C03647=1132.728,344.800,-80.962,-177.361,10.889,149.504
C03648=1132.732,344.553,-80.928,-177.364,10.887,149.505
C03649=1132.736,344.305,-80.893,-177.367,10.884,149.505
C03650=1132.740,344.057,-80.858,-177.370,10.882,149.505
C03651=1132.744,343.810,-80.823,-177.374,10.879,149.505
C03652=1132.748,343.562,-80.789,-177.377,10.877,149.505
C03653=1132.752,343.315,-80.754,-177.380,10.874,149.506
C03654=1132.756,343.067,-80.719,-177.384,10.872,149.506
C03655=1132.760,342.820,-80.685,-177.387,10.869,149.506
C03656=1132.764,342.572,-80.650,-177.390,10.867,149.506
C03657=1132.768,342.325,-80.615,-177.393,10.864,149.506
C03658=1132.771,342.077,-80.581,-177.396,10.862,149.507
C03659=1132.776,341.830,-80.547,-177.400,10.859,149.507
C03660=1132.780,341.582,-80.512,-177.403,10.857,149.507
C03661=1132.784,341.334,-80.478,-177.406,10.854,149.507
C03662=1132.787,341.087,-80.443,-177.409,10.851,149.507
C03663=1132.791,340.840,-80.409,-177.413,10.849,149.508
C03664=1132.795,340.592,-80.374,-177.416,10.847,149.508
C03665=1132.800,340.344,-80.339,-177.419,10.844,149.508
C03666=1132.803,340.097,-80.305,-177.422,10.841,149.508
C03667=1132.808,339.849,-80.271,-177.426,10.839,149.508
C03668=1132.811,339.602,-80.237,-177.429,10.836,149.509
C03669=1132.815,339.354,-80.202,-177.432,10.834,149.509
C03670=1132.819,339.107,-80.168,-177.435,10.832,149.509
C03671=1132.823,338.859,-80.133,-177.438,10.829,149.509
C03672=1132.827,338.612,-80.099,-177.442,10.826,149.509
C03673=1132.831,338.363,-80.065,-177.445,10.824,149.510
C03674=1132.835,338.116,-80.031,-177.448,10.821,149.510
C03675=1132.840,337.868,-79.997,-177.452,10.819,149.510
C03676=1132.843,337.620,-79.963,-177.455,10.816,149.510
C03677=1132.848,337.373,-79.928,-177.458,10.814,149.510
C03678=1132.851,337.125,-79.894,-177.461,10.811,149.511
C03679=1132.855,336.878,-79.860,-177.465,10.809,149.511
C03680=1132.859,336.630,-79.825,-177.468,10.806,149.511
C03681=1132.863,336.383,-79.791,-177.471,10.804,149.511
C03682=1132.867,336.135,-79.758,-177.473,10.802,149.511
C03683=1132.870,335.887,-79.723,-177.477,10.799,149.512
C03684=1132.875,335.674,-79.694,-177.480,10.797,149.512
C03685=1132.877,335.461,-79.664,-177.482,10.795,149.512
C03686=1132.881,335.248,-79.635,-177.486,10.793,149.512
C03687=1132.885,335.034,-79.605,-177.488,10.791,149.512
C03688=1132.888,334.821,-79.576,-177.491,10.788,149.513
C03689=1132.892,334.608,-79.547,-177.494,10.786,149.513
C03690=1132.895,334.395,-79.518,-177.496,10.784,149.513
C03691=1132.899,334.182,-79.489,-177.499,10.782,149.513
C03692=1132.902,333.934,-79.454,-177.503,10.779,149.513
C03693=1132.906,333.687,-79.421,-177.506,10.777,149.513
C03694=1132.911,333.439,-79.387,-177.509,10.774,149.514
C03695=1132.914,333.191,-79.353,-177.512,10.772,149.514
C03696=1132.918,332.943,-79.319,-177.515,10.769,149.514
C03697=1132.923,332.696,-79.285,-177.519,10.767,149.514
C03698=1132.926,332.448,-79.251,-177.522,10.764,149.514
C03699=1132.930,332.200,-79.218,-177.525,10.761,149.515
C03700=1132.934,331.953,-79.184,-177.528,10.759,149.515
C03701=1132.938,331.704,-79.150,-177.531,10.757,149.515
C03702=1132.942,331.457,-79.116,-177.534,10.754,149.515
C03703=1132.946,331.209,-79.083,-177.537,10.752,149.515
C03704=1132.950,330.962,-79.049,-177.541,10.750,149.516
C03705=1132.954,330.714,-79.015,-177.544,10.747,149.516
C03706=1132.958,330.466,-78.981,-177.547,10.744,149.516
C03707=1132.962,330.219,-78.948,-177.550,10.742,149.516
C03708=1132.966,329.972,-78.914,-177.553,10.739,149.516
C03709=1132.970,329.723,-78.880,-177.557,10.737,149.517
C03710=1132.974,329.476,-78.846,-177.560,10.734,149.517
C03711=1132.978,329.228,-78.813,-177.563,10.732,149.517
C03712=1132.982,328.980,-78.779,-177.566,10.729,149.517
C03713=1132.986,328.732,-78.745,-177.569,10.727,149.517
C03714=1132.990,328.485,-78.712,-177.573,10.724,149.517
C03715=1132.994,328.238,-78.678,-177.576,10.722,149.518
C03716=1132.998,327.990,-78.644,-177.579,10.719,149.518
C03717=1133.003,327.742,-78.611,-177.582,10.716,149.518
C03718=1133.006,327.494,-78.577,-177.585,10.714,149.518
C03719=1133.010,327.246,-78.544,-177.589,10.712,149.519
C03720=1133.014,326.999,-78.511,-177.592,10.709,149.519
C03721=1133.018,326.751,-78.478,-177.595,10.706,149.519
C03722=1133.022,326.504,-78.444,-177.598,10.704,149.519
C03723=1133.026,326.256,-78.411,-177.602,10.701,149.519
C03724=1133.030,326.008,-78.377,-177.605,10.699,149.519
C03725=1133.034,325.760,-78.344,-177.608,10.696,149.520
C03726=1133.038,325.512,-78.311,-177.611,10.694,149.520
C03727=1133.042,325.265,-78.277,-177.614,10.691,149.520
C03728=1133.046,325.017,-78.244,-177.617,10.689,149.520
C03729=1133.050,324.770,-78.211,-177.620,10.687,149.521
C03730=1133.054,324.521,-78.177,-177.623,10.684,149.521
C03731=1133.058,324.273,-78.144,-177.626,10.682,149.521
C03732=1133.062,324.026,-78.111,-177.630,10.679,149.521
C03733=1133.066,323.778,-78.078,-177.633,10.676,149.521
C03734=1133.070,323.530,-78.044,-177.636,10.674,149.521
C03735=1133.074,323.283,-78.010,-177.639,10.672,149.522
C03736=1133.078,323.035,-77.977,-177.643,10.669,149.522
C03737=1133.082,322.788,-77.944,-177.646,10.666,149.522
C03738=1133.086,322.540,-77.911,-177.649,10.664,149.522
C03739=1133.090,322.291,-77.877,-177.652,10.661,149.522
C03740=1133.094,322.078,-77.849,-177.655,10.659,149.523
C03741=1133.097,321.865,-77.820,-177.657,10.657,149.523
C03742=1133.100,321.652,-77.793,-177.660,10.655,149.523
C03743=1133.104,321.438,-77.764,-177.663,10.652,149.523
C03744=1133.107,321.225,-77.735,-177.666,10.651,149.523
C03745=1133.111,321.011,-77.707,-177.669,10.648,149.523
C03746=1133.115,320.798,-77.678,-177.671,10.646,149.524
C03747=1133.118,320.585,-77.650,-177.674,10.644,149.524
C03748=1133.123,320.337,-77.617,-177.677,10.642,149.524
C03749=1133.125,320.089,-77.584,-177.680,10.639,149.524
C03750=1133.129,319.841,-77.551,-177.683,10.637,149.524
C03751=1133.134,319.594,-77.518,-177.687,10.634,149.525
C03752=1133.138,319.345,-77.485,-177.690,10.631,149.525
C03753=1133.142,319.098,-77.452,-177.693,10.629,149.525
C03754=1133.146,318.850,-77.420,-177.696,10.626,149.525
C03755=1133.150,318.602,-77.387,-177.699,10.624,149.525
C03756=1133.154,318.355,-77.353,-177.702,10.621,149.525
C03757=1133.158,318.106,-77.321,-177.705,10.618,149.525
C03758=1133.162,317.859,-77.288,-177.709,10.616,149.526
C03759=1133.166,317.611,-77.255,-177.712,10.614,149.526
C03760=1133.170,317.363,-77.222,-177.715,10.611,149.526
C03761=1133.174,317.115,-77.190,-177.718,10.608,149.526
C03762=1133.178,316.868,-77.157,-177.722,10.606,149.527
C03763=1133.182,316.620,-77.124,-177.725,10.603,149.527
C03764=1133.186,316.372,-77.091,-177.728,10.601,149.527
C03765=1133.191,316.125,-77.059,-177.731,10.598,149.527
C03766=1133.195,315.877,-77.026,-177.733,10.596,149.527
C03767=1133.199,315.629,-76.994,-177.737,10.594,149.527
C03768=1133.203,315.381,-76.961,-177.740,10.591,149.528
C03769=1133.207,315.133,-76.929,-177.743,10.589,149.528
C03770=1133.211,314.885,-76.896,-177.746,10.586,149.528
C03771=1133.215,314.638,-76.862,-177.749,10.583,149.528
C03772=1133.219,314.389,-76.831,-177.753,10.581,149.528
C03773=1133.223,314.142,-76.797,-177.756,10.578,149.528
C03774=1133.227,313.894,-76.766,-177.759,10.576,149.529
C03775=1133.231,313.646,-76.732,-177.762,10.573,149.529
C03776=1133.235,313.398,-76.700,-177.765,10.571,149.529
C03777=1133.239,313.151,-76.668,-177.768,10.568,149.529
C03778=1133.244,312.903,-76.635,-177.771,10.565,149.529
C03779=1133.247,312.655,-76.603,-177.775,10.563,149.530
C03780=1133.252,312.407,-76.570,-177.778,10.560,149.530
C03781=1133.256,312.158,-76.538,-177.781,10.558,149.530
C03782=1133.259,311.911,-76.505,-177.784,10.555,149.530
C03783=1133.264,311.663,-76.473,-177.787,10.552,149.530
C03784=1133.268,311.416,-76.441,-177.791,10.550,149.531
C03785=1133.272,311.168,-76.408,-177.794,10.548,149.531
C03786=1133.276,310.920,-76.376,-177.796,10.546,149.531
C03787=1133.280,310.672,-76.343,-177.800,10.543,149.531
C03788=1133.284,310.424,-76.311,-177.802,10.540,149.531
C03789=1133.288,310.175,-76.279,-177.806,10.538,149.532
C03790=1133.292,309.929,-76.247,-177.809,10.536,149.532
C03791=1133.297,309.680,-76.214,-177.812,10.533,149.532
C03792=1133.300,309.432,-76.182,-177.815,10.530,149.532
C03793=1133.305,309.184,-76.150,-177.818,10.528,149.532
C03794=1133.308,308.937,-76.117,-177.822,10.525,149.532
C03795=1133.313,308.689,-76.086,-177.825,10.522,149.533
C03796=1133.316,308.476,-76.058,-177.827,10.521,149.533
C03797=1133.320,308.262,-76.031,-177.830,10.518,149.533
C03798=1133.324,308.048,-76.003,-177.833,10.516,149.533
C03799=1133.327,307.835,-75.975,-177.836,10.514,149.533
C03800=1133.331,307.621,-75.948,-177.838,10.512,149.533
C03801=1133.334,307.408,-75.920,-177.841,10.510,149.534
C03802=1133.338,307.194,-75.892,-177.844,10.507,149.534
C03803=1133.341,306.981,-75.864,-177.846,10.505,149.534
C03804=1133.345,306.733,-75.832,-177.849,10.503,149.534
C03805=1133.349,306.485,-75.800,-177.852,10.500,149.534
C03806=1133.353,306.237,-75.768,-177.856,10.497,149.534
C03807=1133.358,305.989,-75.736,-177.859,10.495,149.535
C03808=1133.361,305.741,-75.704,-177.862,10.492,149.535
C03809=1133.365,305.493,-75.673,-177.865,10.490,149.535
C03810=1133.370,305.245,-75.640,-177.868,10.487,149.535
C03811=1133.374,304.997,-75.609,-177.872,10.485,149.535
C03812=1133.378,304.749,-75.577,-177.874,10.482,149.535
C03813=1133.382,304.501,-75.544,-177.878,10.479,149.536
C03814=1133.386,304.254,-75.513,-177.880,10.477,149.536
C03815=1133.390,304.006,-75.481,-177.883,10.475,149.536
C03816=1133.395,303.757,-75.449,-177.886,10.472,149.536
C03817=1133.399,303.510,-75.417,-177.890,10.470,149.536
C03818=1133.403,303.262,-75.385,-177.893,10.467,149.537
C03819=1133.406,303.014,-75.353,-177.896,10.465,149.537
C03820=1133.412,302.766,-75.322,-177.899,10.462,149.537
C03821=1133.415,302.518,-75.290,-177.902,10.459,149.537
C03822=1133.420,302.270,-75.259,-177.906,10.457,149.537
C03823=1133.423,302.022,-75.227,-177.909,10.454,149.538
C03824=1133.427,301.774,-75.195,-177.912,10.452,149.538
C03825=1133.432,301.526,-75.163,-177.915,10.449,149.538
C03826=1133.436,301.278,-75.132,-177.918,10.447,149.538
C03827=1133.440,301.030,-75.100,-177.921,10.444,149.538
C03828=1133.444,300.782,-75.068,-177.924,10.441,149.538
C03829=1133.448,300.534,-75.037,-177.927,10.439,149.539
C03830=1133.452,300.286,-75.006,-177.930,10.437,149.539
C03831=1133.457,300.038,-74.973,-177.933,10.434,149.539
C03832=1133.461,299.790,-74.942,-177.936,10.432,149.539
C03833=1133.465,299.543,-74.910,-177.939,10.429,149.539
C03834=1133.469,299.294,-74.879,-177.943,10.427,149.540
C03835=1133.473,299.047,-74.847,-177.945,10.424,149.540
C03836=1133.477,298.799,-74.816,-177.949,10.421,149.540
C03837=1133.482,298.551,-74.785,-177.952,10.419,149.540
C03838=1133.485,298.303,-74.753,-177.955,10.416,149.540
C03839=1133.490,298.055,-74.722,-177.958,10.414,149.541
C03840=1133.494,297.807,-74.690,-177.961,10.411,149.541
C03841=1133.497,297.559,-74.659,-177.965,10.409,149.541
C03842=1133.502,297.311,-74.628,-177.968,10.406,149.541
C03843=1133.506,297.063,-74.596,-177.971,10.403,149.541
C03844=1133.510,296.815,-74.565,-177.973,10.401,149.541
C03845=1133.514,296.567,-74.533,-177.977,10.399,149.542
C03846=1133.518,296.319,-74.503,-177.980,10.396,149.542
C03847=1133.522,296.071,-74.471,-177.983,10.394,149.542
C03848=1133.527,295.823,-74.440,-177.986,10.391,149.542
C03849=1133.531,295.575,-74.408,-177.989,10.389,149.542
C03850=1133.535,295.327,-74.377,-177.992,10.386,149.542
C03851=1133.539,295.079,-74.346,-177.995,10.383,149.543
C03852=1133.542,294.865,-74.319,-177.998,10.381,149.543
C03853=1133.546,294.652,-74.292,-178.001,10.379,149.543
C03854=1133.550,294.438,-74.265,-178.003,10.377,149.543
C03855=1133.553,294.224,-74.238,-178.006,10.375,149.543
C03856=1133.557,294.010,-74.211,-178.009,10.372,149.543
C03857=1133.561,293.797,-74.185,-178.011,10.370,149.544
C03858=1133.565,293.583,-74.158,-178.014,10.368,149.544
C03859=1133.568,293.369,-74.131,-178.017,10.366,149.544
C03860=1133.573,293.121,-74.100,-178.019,10.363,149.544
C03861=1133.576,292.874,-74.069,-178.023,10.361,149.544
C03862=1133.580,292.626,-74.038,-178.026,10.358,149.544
C03863=1133.584,292.377,-74.007,-178.029,10.356,149.545
C03864=1133.588,292.130,-73.975,-178.032,10.353,149.545
C03865=1133.592,291.881,-73.944,-178.035,10.350,149.545
C03866=1133.597,291.633,-73.914,-178.038,10.348,149.545
C03867=1133.600,291.385,-73.883,-178.041,10.346,149.545
C03868=1133.605,291.137,-73.852,-178.044,10.343,149.545
C03869=1133.609,290.889,-73.821,-178.047,10.341,149.546
C03870=1133.613,290.641,-73.790,-178.050,10.338,149.546
C03871=1133.618,290.393,-73.759,-178.053,10.335,149.546
C03872=1133.622,290.145,-73.729,-178.056,10.333,149.546
C03873=1133.625,289.897,-73.697,-178.059,10.330,149.546
C03874=1133.630,289.649,-73.666,-178.063,10.328,149.547
C03875=1133.634,289.400,-73.635,-178.066,10.325,149.547
C03876=1133.638,289.153,-73.605,-178.069,10.322,149.547
C03877=1133.643,288.905,-73.574,-178.072,10.320,149.547
C03878=1133.647,288.656,-73.543,-178.075,10.318,149.547
C03879=1133.650,288.408,-73.513,-178.078,10.315,149.547
C03880=1133.655,288.161,-73.482,-178.081,10.313,149.548
C03881=1133.659,287.912,-73.451,-178.084,10.310,149.548
C03882=1133.664,287.664,-73.420,-178.087,10.307,149.548
C03883=1133.668,287.416,-73.390,-178.090,10.305,149.548
C03884=1133.672,287.168,-73.359,-178.093,10.302,149.548
C03885=1133.676,286.920,-73.328,-178.096,10.300,149.549
C03886=1133.680,286.672,-73.298,-178.099,10.297,149.549
C03887=1133.684,286.423,-73.267,-178.103,10.295,149.549
C03888=1133.688,286.176,-73.237,-178.106,10.292,149.549
C03889=1133.693,285.928,-73.206,-178.109,10.289,149.549
C03890=1133.697,285.680,-73.175,-178.111,10.287,149.549
C03891=1133.700,285.431,-73.144,-178.114,10.285,149.550
C03892=1133.705,285.183,-73.114,-178.118,10.282,149.550
C03893=1133.709,284.936,-73.084,-178.121,10.279,149.550
C03894=1133.714,284.688,-73.053,-178.124,10.277,149.550
C03895=1133.718,284.439,-73.022,-178.127,10.274,149.550
C03896=1133.722,284.191,-72.992,-178.130,10.272,149.551
C03897=1133.726,283.943,-72.961,-178.133,10.269,149.551
C03898=1133.730,283.695,-72.931,-178.136,10.267,149.551
C03899=1133.734,283.447,-72.900,-178.139,10.264,149.551
C03900=1133.738,283.198,-72.871,-178.142,10.261,149.551
C03901=1133.743,282.950,-72.840,-178.145,10.259,149.551
C03902=1133.747,282.703,-72.810,-178.148,10.257,149.552
C03903=1133.751,282.454,-72.779,-178.151,10.254,149.552
C03904=1133.755,282.206,-72.749,-178.154,10.252,149.552
C03905=1133.760,281.958,-72.718,-178.158,10.249,149.552
C03906=1133.764,281.710,-72.688,-178.161,10.246,149.552
C03907=1133.768,281.462,-72.657,-178.163,10.244,149.552
C03908=1133.772,281.248,-72.631,-178.167,10.241,149.553
C03909=1133.776,281.034,-72.606,-178.170,10.239,149.553
C03910=1133.779,280.821,-72.579,-178.173,10.236,149.553
C03911=1133.783,280.606,-72.553,-178.176,10.234,149.553
C03912=1133.786,280.393,-72.528,-178.179,10.231,149.553
C03913=1133.790,280.179,-72.501,-178.183,10.228,149.554
C03914=1133.794,279.965,-72.475,-178.185,10.226,149.554
C03915=1133.797,279.751,-72.450,-178.188,10.224,149.554
C03916=1133.801,279.503,-72.419,-178.192,10.221,149.554
C03917=1133.806,279.255,-72.390,-178.195,10.218,149.554
C03918=1133.810,279.007,-72.359,-178.199,10.215,149.555
C03919=1133.814,278.759,-72.329,-178.203,10.213,149.555
C03920=1133.818,278.511,-72.299,-178.206,10.209,149.555
C03921=1133.822,278.262,-72.269,-178.210,10.207,149.555
C03922=1133.827,278.014,-72.239,-178.212,10.204,149.555
C03923=1133.831,277.766,-72.209,-178.216,10.201,149.556
C03924=1133.835,277.518,-72.179,-178.220,10.198,149.556
C03925=1133.839,277.270,-72.149,-178.223,10.195,149.556
C03926=1133.844,277.021,-72.119,-178.227,10.192,149.556
C03927=1133.848,276.774,-72.089,-178.230,10.189,149.557
C03928=1133.852,276.525,-72.060,-178.233,10.187,149.557
C03929=1133.856,276.277,-72.029,-178.237,10.184,149.557
C03930=1133.861,276.029,-72.000,-178.240,10.181,149.557
C03931=1133.865,275.781,-71.970,-178.243,10.178,149.557
C03932=1133.869,275.533,-71.940,-178.246,10.176,149.557
C03933=1133.873,275.284,-71.910,-178.249,10.173,149.557
C03934=1133.877,275.036,-71.880,-178.253,10.170,149.558
C03935=1133.881,274.787,-71.851,-178.256,10.167,149.558
C03936=1133.885,274.540,-71.820,-178.259,10.164,149.558
C03937=1133.889,274.291,-71.791,-178.262,10.161,149.558
C03938=1133.894,274.043,-71.762,-178.265,10.159,149.558
C03939=1133.898,273.795,-71.732,-178.268,10.156,149.558
C03940=1133.903,273.546,-71.702,-178.271,10.153,149.559
C03941=1133.906,273.299,-71.672,-178.274,10.151,149.559
C03942=1133.911,273.050,-71.642,-178.277,10.148,149.559
C03943=1133.915,272.802,-71.613,-178.280,10.146,149.559
C03944=1133.919,272.554,-71.584,-178.283,10.143,149.559
C03945=1133.923,272.306,-71.554,-178.286,10.140,149.559
C03946=1133.927,272.057,-71.525,-178.289,10.137,149.559
C03947=1133.932,271.809,-71.495,-178.292,10.135,149.559
C03948=1133.937,271.561,-71.466,-178.295,10.132,149.560
C03949=1133.941,271.314,-71.435,-178.297,10.130,149.560
C03950=1133.945,271.065,-71.406,-178.300,10.127,149.560
C03951=1133.949,270.817,-71.376,-178.303,10.124,149.560
C03952=1133.954,270.569,-71.347,-178.306,10.121,149.560
C03953=1133.958,270.321,-71.318,-178.309,10.119,149.560
C03954=1133.962,270.072,-71.288,-178.311,10.117,149.560
C03955=1133.966,269.824,-71.259,-178.314,10.114,149.560
C03956=1133.970,269.576,-71.229,-178.317,10.111,149.560
C03957=1133.974,269.327,-71.200,-178.319,10.109,149.561
C03958=1133.979,269.079,-71.170,-178.322,10.107,149.561
C03959=1133.983,268.830,-71.142,-178.325,10.104,149.561
C03960=1133.987,268.582,-71.112,-178.327,10.102,149.561
C03961=1133.992,268.334,-71.083,-178.330,10.099,149.561
C03962=1133.996,268.086,-71.054,-178.333,10.097,149.561
C03963=1134.000,267.838,-71.024,-178.335,10.094,149.561
C03964=1134.003,267.624,-70.999,-178.338,10.092,149.561
C03965=1134.007,267.410,-70.974,-178.340,10.090,149.561
C03966=1134.012,267.196,-70.948,-178.342,10.088,149.561
C03967=1134.015,266.982,-70.923,-178.344,10.086,149.561
C03968=1134.018,266.768,-70.898,-178.346,10.084,149.561
C03969=1134.023,266.554,-70.873,-178.349,10.082,149.562
C03970=1134.026,266.341,-70.847,-178.351,10.080,149.562
C03971=1134.030,266.126,-70.822,-178.353,10.077,149.562
C03972=1134.034,265.878,-70.793,-178.355,10.075,149.562
C03973=1134.039,265.630,-70.764,-178.357,10.073,149.562
C03974=1134.043,265.382,-70.734,-178.360,10.071,149.562
C03975=1134.047,265.133,-70.706,-178.362,10.068,149.562
C03976=1134.051,264.885,-70.677,-178.365,10.066,149.562
C03977=1134.055,264.637,-70.647,-178.367,10.064,149.562
C03978=1134.059,264.388,-70.618,-178.370,10.062,149.562
C03979=1134.064,264.140,-70.590,-178.374,10.058,149.563
C03980=1134.068,263.892,-70.560,-178.378,10.055,149.563
C03981=1134.072,263.644,-70.531,-178.382,10.052,149.563
C03982=1134.077,263.395,-70.502,-178.386,10.049,149.563
C03983=1134.080,263.147,-70.473,-178.390,10.046,149.564
C03984=1134.085,262.899,-70.444,-178.394,10.043,149.564
C03985=1134.090,262.650,-70.415,-178.397,10.039,149.564
C03986=1134.094,262.402,-70.386,-178.401,10.036,149.564
C03987=1134.098,262.154,-70.358,-178.405,10.033,149.565
C03988=1134.102,261.906,-70.329,-178.409,10.029,149.565
C03989=1134.107,261.657,-70.300,-178.413,10.026,149.565
C03990=1134.111,261.409,-70.270,-178.417,10.023,149.565
C03991=1134.115,261.161,-70.243,-178.420,10.019,149.565
C03992=1134.120,260.913,-70.213,-178.424,10.017,149.566
C03993=1134.124,260.664,-70.184,-178.427,10.013,149.566
C03994=1134.127,260.416,-70.156,-178.431,10.010,149.566
C03995=1134.133,260.168,-70.127,-178.434,10.007,149.566
C03996=1134.137,259.919,-70.098,-178.438,10.004,149.566
C03997=1134.140,259.671,-70.070,-178.442,10.001,149.567
C03998=1134.146,259.423,-70.041,-178.445,9.998,149.567
C03999=1134.150,259.174,-70.012,-178.448,9.994,149.567
C04000=1134.154,258.926,-69.984,-178.452,9.992,149.567
C04001=1134.159,258.678,-69.955,-178.455,9.988,149.567
C04002=1134.162,258.430,-69.926,-178.458,9.986,149.567
C04003=1134.167,258.181,-69.898,-178.461,9.983,149.567
C04004=1134.172,257.933,-69.869,-178.465,9.979,149.567
C04005=1134.175,257.685,-69.840,-178.468,9.977,149.568
C04006=1134.180,257.436,-69.812,-178.471,9.974,149.568
C04007=1134.184,257.188,-69.784,-178.474,9.971,149.568
C04008=1134.188,256.939,-69.755,-178.477,9.968,149.568
C04009=1134.192,256.691,-69.726,-178.480,9.965,149.568
C04010=1134.197,256.443,-69.698,-178.483,9.962,149.568
C04011=1134.201,256.194,-69.670,-178.486,9.959,149.568
C04012=1134.206,255.946,-69.641,-178.489,9.956,149.568
C04013=1134.210,255.698,-69.613,-178.488,9.956,149.568
C04014=1134.214,255.450,-69.584,-178.486,9.956,149.567
C04015=1134.218,255.201,-69.556,-178.485,9.955,149.567
C04016=1134.223,254.952,-69.527,-178.484,9.955,149.567
C04017=1134.227,254.705,-69.500,-178.484,9.954,149.566
C04018=1134.231,254.456,-69.471,-178.484,9.953,149.566
C04019=1134.236,254.208,-69.443,-178.484,9.952,149.566
C04020=1134.239,253.993,-69.418,-178.484,9.951,149.566
C04021=1134.243,253.780,-69.393,-178.485,9.950,149.566
C04022=1134.246,253.566,-69.369,-178.486,9.949,149.566
C04023=1134.250,253.352,-69.344,-178.487,9.947,149.566
C04024=1134.254,253.138,-69.320,-178.489,9.946,149.566
C04025=1134.258,252.923,-69.295,-178.490,9.944,149.566
C04026=1134.262,252.709,-69.271,-178.492,9.943,149.566
C04027=1134.266,252.495,-69.246,-178.494,9.941,149.566
C04028=1134.270,252.247,-69.218,-178.496,9.939,149.566
C04029=1134.273,251.998,-69.190,-178.499,9.936,149.566
C04030=1134.278,251.750,-69.162,-178.503,9.934,149.566
C04031=1134.282,251.501,-69.133,-178.506,9.930,149.567
C04032=1134.287,251.253,-69.105,-178.509,9.928,149.567
C04033=1134.291,251.005,-69.077,-178.514,9.924,149.567
C04034=1134.296,250.757,-69.049,-178.518,9.921,149.568
C04035=1134.300,250.508,-69.020,-178.523,9.917,149.568
C04036=1134.304,250.260,-68.993,-178.528,9.914,149.568
C04037=1134.309,250.011,-68.964,-178.533,9.910,149.569
C04038=1134.313,249.763,-68.936,-178.539,9.906,149.569
C04039=1134.317,249.515,-68.908,-178.545,9.901,149.570
C04040=1134.322,249.267,-68.880,-178.551,9.897,149.570
C04041=1134.326,249.018,-68.851,-178.558,9.891,149.571
C04042=1134.330,248.770,-68.824,-178.564,9.887,149.571
C04043=1134.334,248.521,-68.796,-178.572,9.881,149.572
C04044=1134.339,248.273,-68.768,-178.579,9.876,149.573
C04045=1134.343,248.024,-68.740,-178.586,9.870,149.573
C04046=1134.347,247.776,-68.712,-178.595,9.864,149.574
C04047=1134.352,247.528,-68.685,-178.603,9.858,149.575
C04048=1134.356,247.279,-68.657,-178.607,9.854,149.575
C04049=1134.361,247.031,-68.628,-178.608,9.852,149.575
C04050=1134.365,246.782,-68.601,-178.609,9.850,149.574
C04051=1134.369,246.534,-68.573,-178.610,9.848,149.574
C04052=1134.374,246.285,-68.546,-178.611,9.846,149.574
C04053=1134.377,246.037,-68.518,-178.613,9.844,149.574
C04054=1134.382,245.789,-68.490,-178.614,9.842,149.574
C04055=1134.386,245.540,-68.463,-178.614,9.840,149.573
C04056=1134.391,245.292,-68.434,-178.616,9.838,149.573
C04057=1134.396,245.043,-68.407,-178.617,9.836,149.573
C04058=1134.400,244.795,-68.380,-178.618,9.834,149.573
C04059=1134.404,244.546,-68.352,-178.619,9.832,149.573
C04060=1134.408,244.298,-68.324,-178.621,9.830,149.573
C04061=1134.412,244.049,-68.297,-178.622,9.828,149.573
C04062=1134.417,243.801,-68.269,-178.624,9.826,149.573
C04063=1134.421,243.553,-68.241,-178.625,9.824,149.573
C04064=1134.425,243.304,-68.214,-178.627,9.822,149.572
C04065=1134.430,243.056,-68.186,-178.629,9.819,149.572
C04066=1134.434,242.808,-68.159,-178.630,9.818,149.572
C04067=1134.438,242.559,-68.131,-178.632,9.816,149.572
C04068=1134.443,242.311,-68.104,-178.634,9.813,149.572
C04069=1134.447,242.062,-68.077,-178.636,9.811,149.572
C04070=1134.452,241.814,-68.048,-178.638,9.809,149.572
C04071=1134.456,241.565,-68.021,-178.640,9.806,149.572
C04072=1134.461,241.317,-67.993,-178.642,9.804,149.572
C04073=1134.465,241.068,-67.966,-178.644,9.802,149.572
C04074=1134.469,240.820,-67.938,-178.646,9.800,149.572
C04075=1134.474,240.571,-67.911,-178.648,9.797,149.572
C04076=1134.478,240.291,-67.880,-178.650,9.795,149.572
C04077=1134.484,240.010,-67.849,-178.653,9.792,149.572
C04078=1134.488,239.730,-67.819,-178.655,9.789,149.572
C04079=1134.493,239.450,-67.787,-178.657,9.787,149.572
C04080=1134.498,239.201,-67.760,-178.660,9.784,149.572
C04081=1134.502,238.952,-67.733,-178.662,9.782,149.572
C04082=1134.506,238.704,-67.705,-178.665,9.780,149.572
C04083=1134.511,238.456,-67.678,-178.667,9.777,149.573
C04084=1134.516,238.207,-67.651,-178.670,9.774,149.572
C04085=1134.520,237.958,-67.623,-178.672,9.772,149.573
C04086=1134.524,237.710,-67.596,-178.675,9.769,149.573
C04087=1134.529,237.462,-67.569,-178.677,9.767,149.573
C04088=1134.533,237.213,-67.541,-178.680,9.764,149.573
C04089=1134.536,236.965,-67.514,-178.683,9.762,149.573
C04090=1134.541,236.716,-67.487,-178.686,9.759,149.573
C04091=1134.546,236.468,-67.460,-178.689,9.756,149.573
C04092=1134.550,236.219,-67.433,-178.692,9.753,149.573
C04093=1134.554,235.970,-67.405,-178.695,9.751,149.573
C04094=1134.559,235.722,-67.378,-178.698,9.748,149.574
C04095=1134.563,235.474,-67.350,-178.701,9.745,149.574
C04096=1134.567,235.226,-67.324,-178.704,9.742,149.574
C04097=1134.572,234.977,-67.297,-178.707,9.740,149.574
C04098=1134.577,234.729,-67.270,-178.710,9.737,149.574
C04099=1134.581,234.480,-67.242,-178.713,9.734,149.574
C04100=1134.585,234.231,-67.215,-178.716,9.731,149.574
C04101=1134.589,233.983,-67.189,-178.719,9.728,149.574
C04102=1134.594,233.734,-67.162,-178.723,9.725,149.575
C04103=1134.598,233.486,-67.135,-178.726,9.722,149.575
C04104=1134.603,233.237,-67.108,-178.730,9.718,149.575
C04105=1134.606,232.988,-67.081,-178.733,9.716,149.575
C04106=1134.611,232.740,-67.054,-178.737,9.713,149.575
C04107=1134.616,232.491,-67.027,-178.740,9.709,149.576
C04108=1134.635,231.404,-66.912,-177.831,7.908,148.890
C04109=1134.639,231.186,-66.889,-177.834,7.905,148.890
C04110=1134.643,230.967,-66.866,-177.836,7.903,148.890
C04111=1134.647,230.748,-66.843,-177.839,7.900,148.890
C04112=1134.651,230.500,-66.817,-177.842,7.897,148.890
C04113=1134.656,230.251,-66.790,-177.845,7.894,148.890
C04114=1134.660,230.003,-66.764,-177.847,7.891,148.890
C04115=1134.664,229.754,-66.738,-177.850,7.888,148.890
C04116=1134.669,229.506,-66.711,-177.853,7.885,148.891
C04117=1134.673,229.257,-66.685,-177.856,7.882,148.891
C04118=1134.678,229.008,-66.658,-177.858,7.880,148.891
C04119=1134.682,228.760,-66.632,-177.861,7.877,148.891
C04120=1134.687,228.512,-66.606,-177.864,7.874,148.891
C04121=1134.692,228.263,-66.580,-177.866,7.872,148.891
C04122=1134.696,228.014,-66.554,-177.869,7.869,148.891
C04123=1134.700,227.766,-66.528,-177.872,7.866,148.891
C04124=1134.705,227.517,-66.501,-177.875,7.863,148.891
C04125=1134.709,227.268,-66.476,-177.878,7.860,148.892
C04126=1134.713,227.020,-66.449,-177.881,7.857,148.892
C04127=1134.718,226.771,-66.423,-177.884,7.854,148.892
C04128=1134.723,226.523,-66.397,-177.887,7.852,148.892
C04129=1134.727,226.274,-66.371,-177.889,7.849,148.892
C04130=1134.732,226.025,-66.345,-177.892,7.846,148.892
C04131=1134.736,225.777,-66.319,-177.895,7.843,148.892
C04132=1134.740,225.528,-66.293,-177.898,7.840,148.892
C04133=1134.745,225.280,-66.267,-177.901,7.837,148.892
C04134=1134.749,225.031,-66.241,-177.903,7.834,148.892
C04135=1134.754,224.782,-66.215,-177.906,7.832,148.893
C04136=1134.758,224.534,-66.189,-177.909,7.830,148.893
C04137=1134.762,224.285,-66.163,-177.912,7.827,148.893
C04138=1134.767,224.037,-66.137,-177.915,7.824,148.893
C04139=1134.772,223.788,-66.111,-177.917,7.821,148.893
C04140=1134.776,223.539,-66.085,-177.920,7.818,148.893
C04141=1134.780,223.291,-66.059,-177.923,7.815,148.893
C04142=1134.784,223.042,-66.034,-177.926,7.812,148.893
C04143=1134.789,222.794,-66.008,-177.929,7.809,148.893
C04144=1134.794,222.545,-65.982,-177.931,7.806,148.894
C04145=1134.798,222.296,-65.956,-177.935,7.804,148.894
C04146=1134.802,222.048,-65.930,-177.937,7.801,148.894
C04147=1134.807,221.799,-65.904,-177.940,7.799,148.894
C04148=1134.811,221.551,-65.879,-177.943,7.796,148.894
C04149=1134.816,221.302,-65.853,-177.945,7.793,148.894
C04150=1134.820,221.054,-65.828,-177.948,7.790,148.894
C04151=1134.825,220.805,-65.802,-177.951,7.787,148.894
C04152=1134.829,220.556,-65.776,-177.954,7.785,148.895
C04153=1134.834,220.307,-65.750,-177.957,7.782,148.895
C04154=1134.839,220.059,-65.724,-177.960,7.779,148.895
C04155=1134.843,219.810,-65.699,-177.963,7.776,148.895
C04156=1134.847,219.561,-65.673,-177.965,7.774,148.895
C04157=1134.852,219.313,-65.648,-177.968,7.771,148.895
C04158=1134.856,219.064,-65.622,-177.971,7.768,148.895
C04159=1134.861,218.815,-65.597,-177.974,7.765,148.896
C04160=1134.865,218.567,-65.571,-177.977,7.763,148.896
C04161=1134.870,218.318,-65.545,-177.979,7.760,148.896
C04162=1134.874,218.069,-65.520,-177.982,7.757,148.896
C04163=1134.879,217.821,-65.494,-177.985,7.754,148.896
C04164=1134.883,217.572,-65.469,-177.988,7.751,148.896
C04165=1134.887,217.323,-65.444,-177.991,7.749,148.897
C04166=1134.892,217.075,-65.418,-177.993,7.746,148.897
C04167=1134.897,216.826,-65.392,-177.996,7.743,148.897
C04168=1134.901,216.577,-65.367,-177.999,7.741,148.897
C04169=1134.905,216.329,-65.343,-178.002,7.738,148.897
C04170=1134.909,216.080,-65.317,-178.005,7.735,148.897
C04171=1134.914,215.832,-65.291,-178.008,7.732,148.897
C04172=1134.918,215.583,-65.266,-178.010,7.730,148.897
C04173=1134.923,215.334,-65.241,-178.013,7.727,148.898
C04174=1134.928,215.086,-65.215,-178.016,7.724,148.898
C04175=1134.932,214.837,-65.190,-178.019,7.722,148.898
C04176=1134.937,214.588,-65.165,-178.022,7.719,148.898
C04177=1134.941,214.339,-65.139,-178.025,7.716,148.898
C04178=1134.946,214.090,-65.113,-178.027,7.713,148.898
C04179=1134.950,213.842,-65.089,-178.030,7.711,148.898
C04180=1134.954,213.593,-65.064,-178.033,7.708,148.899
C04181=1134.959,213.344,-65.039,-178.036,7.706,148.899
C04182=1134.964,213.096,-65.013,-178.039,7.703,148.899
C04183=1134.968,212.848,-64.988,-178.041,7.700,148.899
C04184=1134.972,212.598,-64.963,-178.045,7.697,148.899
C04185=1134.977,212.350,-64.938,-178.047,7.695,148.899
C04186=1134.982,212.101,-64.913,-178.050,7.692,148.900
C04187=1134.986,211.853,-64.887,-178.052,7.689,148.900
C04188=1134.991,211.603,-64.862,-178.056,7.687,148.900
C04189=1134.995,211.356,-64.838,-178.059,7.684,148.900
C04190=1135.000,211.106,-64.813,-178.061,7.681,148.900
C04191=1135.004,210.858,-64.787,-178.064,7.679,148.900
C04192=1135.009,210.609,-64.762,-178.067,7.676,148.901
C04193=1135.013,210.361,-64.737,-178.070,7.673,148.901
C04194=1135.017,210.111,-64.712,-178.073,7.671,148.901
C04195=1135.023,209.863,-64.688,-178.075,7.668,148.901
C04196=1135.027,209.592,-64.661,-178.079,7.665,148.901
C04197=1135.031,209.322,-64.633,-178.081,7.662,148.901
C04198=1135.037,209.051,-64.606,-178.084,7.659,148.902
C04199=1135.042,208.780,-64.578,-178.088,7.657,148.902
C04200=1135.046,208.532,-64.554,-178.090,7.654,148.902
C04201=1135.051,208.282,-64.529,-178.093,7.651,148.902
C04202=1135.056,208.034,-64.504,-178.096,7.648,148.902
C04203=1135.059,207.785,-64.480,-178.099,7.646,148.902
C04204=1135.065,207.536,-64.455,-178.101,7.643,148.903
C04205=1135.070,207.288,-64.430,-178.105,7.641,148.903
C04206=1135.073,207.039,-64.405,-178.108,7.638,148.903
C04207=1135.078,206.790,-64.380,-178.110,7.635,148.903
C04208=1135.082,206.541,-64.356,-178.113,7.633,148.903
C04209=1135.087,206.293,-64.331,-178.116,7.630,148.904
C04210=1135.092,206.045,-64.306,-178.119,7.628,148.904
C04211=1135.096,205.795,-64.281,-178.122,7.625,148.904
C04212=1135.101,205.547,-64.257,-178.125,7.622,148.904
C04213=1135.105,205.298,-64.232,-178.127,7.620,148.904
C04214=1135.110,205.049,-64.208,-178.130,7.617,148.904
C04215=1135.114,204.801,-64.183,-178.133,7.615,148.905
C04216=1135.119,204.552,-64.158,-178.136,7.612,148.905
C04217=1135.123,204.303,-64.134,-178.138,7.610,148.905
C04218=1135.128,204.055,-64.109,-178.141,7.607,148.905
C04219=1135.132,203.805,-64.085,-178.144,7.604,148.905
C04220=1135.137,203.557,-64.060,-178.147,7.601,148.905
C04221=1135.141,203.308,-64.036,-178.149,7.599,148.906
C04222=1135.146,203.059,-64.011,-178.153,7.597,148.906
C04223=1135.150,202.810,-63.987,-178.155,7.594,148.906
C04224=1135.155,202.562,-63.962,-178.158,7.591,148.906
C04225=1135.159,202.313,-63.938,-178.161,7.589,148.906
C04226=1135.164,202.064,-63.913,-178.164,7.586,148.907
C04227=1135.169,201.815,-63.889,-178.167,7.584,148.907
C04228=1135.173,201.566,-63.864,-178.170,7.581,148.907
C04229=1135.178,201.318,-63.840,-178.172,7.579,148.907
C04230=1135.182,201.069,-63.816,-178.175,7.576,148.908
C04231=1135.187,200.820,-63.791,-178.178,7.573,148.908
C04232=1135.191,200.571,-63.767,-178.181,7.570,148.908
C04233=1135.195,200.323,-63.743,-178.184,7.569,148.908
C04234=1135.201,200.074,-63.718,-178.186,7.566,148.908
C04235=1135.205,199.826,-63.694,-178.189,7.563,148.908
C04236=1135.209,199.576,-63.669,-178.193,7.560,148.909
C04237=1135.214,199.327,-63.645,-178.195,7.558,148.909
C04238=1135.219,199.079,-63.621,-178.198,7.556,148.909
C04239=1135.224,198.830,-63.597,-178.201,7.553,148.909
C04240=1135.227,198.581,-63.572,-178.203,7.551,148.909
C04241=1135.232,198.333,-63.548,-178.206,7.548,148.910
C04242=1135.236,198.084,-63.524,-178.209,7.545,148.910
C04243=1135.242,197.835,-63.500,-178.212,7.542,148.910
C04244=1135.245,197.586,-63.476,-178.215,7.541,148.910
C04245=1135.250,197.337,-63.452,-178.218,7.538,148.910
C04246=1135.255,197.089,-63.427,-178.221,7.535,148.911
C04247=1135.260,196.840,-63.404,-178.223,7.533,148.911
C04248=1135.264,196.591,-63.380,-178.226,7.530,148.911
C04249=1135.268,196.342,-63.355,-178.229,7.528,148.911
C04250=1135.273,196.093,-63.331,-178.232,7.525,148.911
C04251=1135.278,195.844,-63.307,-178.235,7.523,148.912
C04252=1135.282,195.596,-63.283,-178.237,7.520,148.912
C04253=1135.287,195.347,-63.260,-178.240,7.517,148.912
C04254=1135.291,195.099,-63.236,-178.243,7.516,148.912
C04255=1135.296,194.850,-63.211,-178.246,7.513,148.912
C04256=1135.300,194.600,-63.187,-178.249,7.510,148.913
C04257=1135.305,194.352,-63.163,-178.251,7.508,148.913
C04258=1135.310,194.103,-63.140,-178.255,7.506,148.913
C04259=1135.314,193.854,-63.116,-178.257,7.503,148.913
C04260=1135.318,193.606,-63.092,-178.260,7.501,148.914
C04261=1135.324,193.356,-63.068,-178.263,7.498,148.914
C04262=1135.328,193.108,-63.044,-178.266,7.495,148.914
C04263=1135.333,192.859,-63.020,-178.268,7.493,148.914
C04264=1135.337,192.610,-62.996,-178.271,7.490,148.914
C04265=1135.341,192.361,-62.972,-178.275,7.488,148.915
C04266=1135.346,192.112,-62.948,-178.277,7.486,148.915
C04267=1135.350,191.863,-62.925,-178.280,7.483,148.915
C04268=1135.355,191.615,-62.901,-178.283,7.480,148.915
C04269=1135.360,191.366,-62.878,-178.285,7.478,148.915
C04270=1135.364,191.118,-62.853,-178.288,7.476,148.916
C04271=1135.369,190.868,-62.829,-178.291,7.473,148.916
C04272=1135.374,190.619,-62.806,-178.294,7.471,148.916
C04273=1135.378,190.371,-62.782,-178.297,7.468,148.916
C04274=1135.383,190.122,-62.759,-178.300,7.466,148.917
C04275=1135.388,189.873,-62.735,-178.302,7.464,148.917
C04276=1135.392,189.624,-62.711,-178.306,7.461,148.917
C04277=1135.397,189.375,-62.688,-178.308,7.458,148.917
C04278=1135.401,189.127,-62.664,-178.311,7.457,148.918
C04279=1135.406,188.878,-62.640,-178.314,7.454,148.918
C04280=1135.411,188.629,-62.617,-178.317,7.451,148.918
C04281=1135.415,188.380,-62.594,-178.319,7.449,148.918
C04282=1135.420,188.131,-62.570,-178.322,7.446,148.918
C04283=1135.425,187.882,-62.546,-178.326,7.444,148.919
C04284=1135.429,187.633,-62.523,-178.328,7.442,148.919
C04285=1135.434,187.384,-62.500,-178.331,7.439,148.919
C04286=1135.438,187.136,-62.476,-178.333,7.437,148.919
C04287=1135.442,186.887,-62.453,-178.337,7.434,148.920
C04288=1135.447,186.638,-62.429,-178.339,7.432,148.920
C04289=1135.452,186.389,-62.406,-178.342,7.430,148.920
C04290=1135.456,186.140,-62.383,-178.345,7.427,148.920
C04291=1135.461,185.892,-62.359,-178.348,7.424,148.921
C04292=1135.465,185.643,-62.335,-178.350,7.422,148.921
C04293=1135.470,185.394,-62.312,-178.354,7.420,148.921
C04294=1135.475,185.144,-62.289,-178.356,7.418,148.921
C04295=1135.479,184.896,-62.266,-178.359,7.415,148.922
C04296=1135.484,184.647,-62.242,-178.362,7.412,148.922
C04297=1135.488,184.398,-62.219,-178.365,7.411,148.922
C04298=1135.493,184.149,-62.196,-178.368,7.408,148.922
C04299=1135.497,183.900,-62.172,-178.370,7.406,148.923
C04300=1135.503,183.630,-62.147,-178.374,7.403,148.923
C04301=1135.507,183.361,-62.122,-178.376,7.400,148.923
C04302=1135.513,183.091,-62.097,-178.380,7.398,148.923
C04303=1135.518,182.822,-62.071,-178.383,7.395,148.924
C04304=1135.522,182.573,-62.048,-178.386,7.393,148.924
C04305=1135.526,182.324,-62.025,-178.388,7.391,148.924
C04306=1135.531,182.075,-62.002,-178.391,7.388,148.924
C04307=1135.536,181.826,-61.979,-178.394,7.386,148.925
C04308=1135.541,181.577,-61.956,-178.397,7.383,148.925
C04309=1135.545,181.329,-61.933,-178.400,7.382,148.925
C04310=1135.550,181.080,-61.910,-178.403,7.379,148.926
C04311=1135.555,180.831,-61.887,-178.406,7.376,148.926
C04312=1135.559,180.582,-61.863,-178.408,7.374,148.926
C04313=1135.563,180.333,-61.841,-178.411,7.372,148.926
C04314=1135.568,180.084,-61.817,-178.414,7.370,148.927
C04315=1135.573,179.835,-61.794,-178.417,7.367,148.927
C04316=1135.577,179.587,-61.772,-178.419,7.365,148.927
C04317=1135.582,179.337,-61.749,-178.422,7.362,148.927
C04318=1135.587,179.088,-61.726,-178.426,7.360,148.928
C04319=1135.591,178.839,-61.703,-178.428,7.358,148.928
C04320=1135.596,178.590,-61.679,-178.431,7.355,148.928
C04321=1135.600,178.342,-61.657,-178.434,7.353,148.928
C04322=1135.605,178.093,-61.634,-178.437,7.351,148.929
C04323=1135.610,177.844,-61.611,-178.439,7.349,148.929
C04324=1135.614,177.595,-61.588,-178.442,7.346,148.929
C04325=1135.619,177.346,-61.565,-178.445,7.344,148.929
C04326=1135.623,177.097,-61.543,-178.448,7.342,148.930
C04327=1135.628,176.848,-61.520,-178.451,7.339,148.930
C04328=1135.633,176.599,-61.496,-178.454,7.337,148.930
C04329=1135.637,176.350,-61.474,-178.456,7.334,148.930
C04330=1135.642,176.101,-61.451,-178.459,7.333,148.931
C04331=1135.646,175.853,-61.429,-178.462,7.330,148.931
C04332=1135.651,175.603,-61.406,-178.465,7.328,148.931
C04333=1135.656,175.355,-61.384,-178.468,7.325,148.932
C04334=1135.661,175.106,-61.360,-178.470,7.323,148.932
C04335=1135.665,174.857,-61.338,-178.473,7.321,148.932
C04336=1135.670,174.608,-61.315,-178.476,7.319,148.932
C04337=1135.674,174.359,-61.293,-178.479,7.316,148.933
C04338=1135.679,174.110,-61.270,-178.482,7.314,148.933
C04339=1135.683,173.861,-61.247,-178.485,7.312,148.933
C04340=1135.689,173.612,-61.225,-178.487,7.310,148.933
C04341=1135.693,173.364,-61.202,-178.491,7.307,148.934
C04342=1135.698,173.114,-61.179,-178.493,7.305,148.934
C04343=1135.702,172.866,-61.157,-178.496,7.303,148.934
C04344=1135.707,172.616,-61.134,-178.499,7.301,148.935
C04345=1135.711,172.368,-61.112,-178.502,7.298,148.935
C04346=1135.717,172.119,-61.089,-178.504,7.296,148.935
C04347=1135.721,171.870,-61.067,-178.507,7.294,148.935
C04348=1135.725,171.621,-61.044,-178.510,7.292,148.936
C04349=1135.731,171.372,-61.022,-178.513,7.289,148.936
C04350=1135.735,171.123,-60.999,-178.515,7.287,148.936
C04351=1135.740,170.873,-60.977,-178.519,7.285,148.937
C04352=1135.744,170.625,-60.954,-178.521,7.283,148.937
C04353=1135.748,170.376,-60.932,-178.524,7.280,148.937
C04354=1135.753,170.126,-60.910,-178.527,7.278,148.937
C04355=1135.758,169.878,-60.887,-178.530,7.276,148.938
C04356=1135.762,169.629,-60.865,-178.532,7.274,148.938
C04357=1135.768,169.380,-60.843,-178.536,7.271,148.938
C04358=1135.772,169.131,-60.820,-178.538,7.270,148.939
C04359=1135.776,168.882,-60.798,-178.541,7.267,148.939
C04360=1135.782,168.633,-60.776,-178.544,7.265,148.939
C04361=1135.786,168.384,-60.753,-178.547,7.262,148.939
C04362=1135.791,168.136,-60.731,-178.550,7.260,148.940
C04363=1135.796,167.886,-60.709,-178.553,7.258,148.940
C04364=1135.800,167.637,-60.687,-178.556,7.256,148.940
C04365=1135.804,167.388,-60.664,-178.558,7.253,148.940
C04366=1135.809,167.140,-60.643,-178.561,7.252,148.941
C04367=1135.814,166.890,-60.620,-178.564,7.249,148.941
C04368=1135.819,166.641,-60.598,-178.567,7.247,148.941
C04369=1135.823,166.393,-60.576,-178.569,7.245,148.942
C04370=1135.827,166.143,-60.554,-178.573,7.243,148.942
C04371=1135.833,165.895,-60.531,-178.575,7.241,148.942
C04372=1135.837,165.645,-60.509,-178.578,7.238,148.943
C04373=1135.842,165.397,-60.488,-178.581,7.236,148.943
C04374=1135.846,165.147,-60.465,-178.584,7.234,148.943
C04375=1135.851,164.899,-60.444,-178.586,7.232,148.944
C04376=1135.856,164.650,-60.420,-178.590,7.229,148.944
C04377=1135.861,164.401,-60.399,-178.592,7.227,148.944
C04378=1135.865,164.152,-60.377,-178.595,7.225,148.944
C04379=1135.870,163.903,-60.355,-178.598,7.223,148.945
C04380=1135.874,163.654,-60.333,-178.601,7.221,148.945
C04381=1135.879,163.405,-60.311,-178.603,7.218,148.945
C04382=1135.883,163.156,-60.289,-178.606,7.217,148.946
C04383=1135.888,162.907,-60.268,-178.609,7.214,148.946
C04384=1135.893,162.657,-60.245,-178.612,7.212,148.946
C04385=1135.898,162.409,-60.223,-178.615,7.210,148.947
C04386=1135.903,162.160,-60.202,-178.618,7.208,148.947
C04387=1135.907,161.911,-60.179,-178.620,7.206,148.947
C04388=1135.912,161.662,-60.158,-178.623,7.203,148.947
C04389=1135.916,161.413,-60.136,-178.626,7.202,148.948
C04390=1135.921,161.164,-60.114,-178.629,7.199,148.948
C04391=1135.926,160.915,-60.092,-178.632,7.197,148.948
C04392=1135.931,160.665,-60.071,-178.634,7.195,148.949
C04393=1135.935,160.416,-60.049,-178.638,7.193,148.949
C04394=1135.940,160.167,-60.027,-178.640,7.191,148.949
C04395=1135.945,159.919,-60.006,-178.643,7.188,148.950
C04396=1135.949,159.670,-59.984,-178.646,7.186,148.950
C04397=1135.954,159.421,-59.962,-178.648,7.185,148.950
C04398=1135.958,159.172,-59.940,-178.652,7.182,148.951
C04399=1135.963,158.923,-59.918,-178.654,7.180,148.951
C04400=1135.968,158.674,-59.897,-178.657,7.178,148.951
C04401=1135.972,158.424,-59.875,-178.660,7.176,148.952
C04402=1135.977,158.176,-59.853,-178.663,7.174,148.952
C04403=1135.982,157.927,-59.832,-178.666,7.171,148.952
C04404=1135.988,157.658,-59.808,-178.669,7.169,148.952
C04405=1135.992,157.389,-59.786,-178.672,7.167,148.953
C04406=1135.998,157.120,-59.762,-178.675,7.165,148.953
C04407=1136.002,156.851,-59.739,-178.678,7.163,148.954
C04408=1136.007,156.601,-59.717,-178.681,7.160,148.954
C04409=1136.012,156.352,-59.696,-178.683,7.158,148.954
C04410=1136.017,156.104,-59.674,-178.686,7.156,148.954
C04411=1136.021,155.855,-59.652,-178.689,7.154,148.955
C04412=1136.026,155.605,-59.631,-178.692,7.152,148.955
C04413=1136.031,155.356,-59.609,-178.695,7.150,148.956
C04414=1136.035,155.108,-59.588,-178.697,7.148,148.956
C04415=1136.040,154.858,-59.567,-178.700,7.146,148.956
C04416=1136.044,154.609,-59.545,-178.703,7.144,148.957
C04417=1136.049,154.361,-59.524,-178.706,7.142,148.957
C04418=1136.054,154.111,-59.502,-178.709,7.139,148.957
C04419=1136.059,153.862,-59.481,-178.712,7.137,148.957
C04420=1136.063,153.613,-59.460,-178.714,7.136,148.958
C04421=1136.068,153.365,-59.439,-178.718,7.133,148.958
C04422=1136.073,153.115,-59.417,-178.720,7.131,148.959
C04423=1136.078,152.866,-59.396,-178.723,7.129,148.959
C04424=1136.083,152.617,-59.375,-178.726,7.127,148.959
C04425=1136.087,152.368,-59.354,-178.729,7.125,148.959
C04426=1136.091,152.118,-59.332,-178.731,7.123,148.960
C04427=1136.096,151.870,-59.311,-178.735,7.121,148.960
C04428=1136.101,151.621,-59.290,-178.737,7.119,148.960
C04429=1136.106,151.372,-59.268,-178.740,7.117,148.961
C04430=1136.111,151.123,-59.247,-178.743,7.115,148.961
C04431=1136.115,150.874,-59.225,-178.746,7.113,148.962
C04432=1136.120,150.624,-59.204,-178.748,7.111,148.962
C04433=1136.124,150.376,-59.183,-178.751,7.108,148.962
C04434=1136.130,150.127,-59.162,-178.754,7.107,148.962
C04435=1136.135,149.877,-59.141,-178.757,7.105,148.963
C04436=1136.139,149.628,-59.119,-178.760,7.102,148.963
C04437=1136.143,149.379,-59.099,-178.763,7.101,148.964
C04438=1136.149,149.130,-59.078,-178.765,7.099,148.964
C04439=1136.153,148.881,-59.056,-178.768,7.096,148.964
C04440=1136.158,148.632,-59.036,-178.771,7.094,148.964
C04441=1136.163,148.383,-59.015,-178.774,7.093,148.965
C04442=1136.167,148.134,-58.994,-178.776,7.091,148.965
C04443=1136.172,147.885,-58.973,-178.780,7.088,148.966
C04444=1136.177,147.636,-58.952,-178.782,7.086,148.966
C04445=1136.181,147.387,-58.931,-178.785,7.085,148.966
C04446=1136.186,147.138,-58.910,-178.788,7.082,148.967
C04447=1136.191,146.889,-58.889,-178.791,7.081,148.967
C04448=1136.196,146.640,-58.868,-178.793,7.079,148.967
C04449=1136.200,146.390,-58.847,-178.797,7.076,148.968
C04450=1136.205,146.141,-58.826,-178.799,7.074,148.968
C04451=1136.210,145.892,-58.805,-178.802,7.073,148.968
C04452=1136.214,145.643,-58.785,-178.804,7.071,148.969
C04453=1136.219,145.394,-58.764,-178.808,7.068,148.969
C04454=1136.225,145.145,-58.743,-178.810,7.067,148.969
C04455=1136.229,144.896,-58.722,-178.813,7.065,148.970
C04456=1136.234,144.647,-58.701,-178.816,7.062,148.970
C04457=1136.238,144.398,-58.680,-178.819,7.060,148.970
C04458=1136.243,144.149,-58.659,-178.821,7.059,148.971
C04459=1136.247,143.899,-58.638,-178.824,7.057,148.971
C04460=1136.252,143.650,-58.617,-178.827,7.054,148.971
C04461=1136.257,143.401,-58.597,-178.830,7.053,148.972
C04462=1136.262,143.152,-58.576,-178.833,7.051,148.972
C04463=1136.267,142.903,-58.556,-178.836,7.049,148.973
C04464=1136.271,142.654,-58.535,-178.838,7.046,148.973
C04465=1136.276,142.405,-58.514,-178.841,7.045,148.973
C04466=1136.281,142.156,-58.494,-178.844,7.043,148.974
C04467=1136.286,141.906,-58.473,-178.847,7.041,148.974
C04468=1136.290,141.657,-58.453,-178.850,7.039,148.974
C04469=1136.295,141.408,-58.432,-178.853,7.037,148.975
C04470=1136.300,141.159,-58.411,-178.855,7.035,148.975
C04471=1136.304,140.910,-58.391,-178.858,7.033,148.975
C04472=1136.309,140.661,-58.370,-178.861,7.031,148.976
C04473=1136.314,140.412,-58.350,-178.864,7.029,148.976
C04474=1136.319,140.163,-58.329,-178.866,7.028,148.976
C04475=1136.323,139.914,-58.308,-178.870,7.025,148.977
C04476=1136.328,139.665,-58.288,-178.872,7.023,148.977
C04477=1136.333,139.416,-58.267,-178.875,7.022,148.978
C04478=1136.337,139.167,-58.247,-178.878,7.020,148.978
C04479=1136.342,138.918,-58.226,-178.881,7.017,148.978
C04480=1136.347,138.668,-58.206,-178.883,7.015,148.979
C04481=1136.352,138.419,-58.186,-178.886,7.014,148.979
C04482=1136.356,138.170,-58.165,-178.889,7.012,148.979
C04483=1136.361,137.921,-58.144,-178.891,7.010,148.980
C04484=1136.366,137.672,-58.124,-178.895,7.008,148.980
C04485=1136.371,137.422,-58.104,-178.898,7.006,148.980
C04486=1136.375,137.173,-58.084,-178.900,7.004,148.981
C04487=1136.381,136.925,-58.063,-178.903,7.003,148.981
C04488=1136.385,136.676,-58.043,-178.906,7.000,148.982
C04489=1136.390,136.427,-58.023,-178.909,6.998,148.982
C04490=1136.395,136.177,-58.002,-178.912,6.997,148.982
C04491=1136.400,135.928,-57.982,-178.914,6.995,148.983
C04492=1136.404,135.679,-57.962,-178.917,6.993,148.983
C04493=1136.409,135.429,-57.942,-178.920,6.991,148.983
C04494=1136.414,135.180,-57.921,-178.923,6.989,148.984
C04495=1136.418,134.931,-57.901,-178.925,6.987,148.984
C04496=1136.423,134.682,-57.881,-178.928,6.985,148.985
C04497=1136.428,134.433,-57.861,-178.931,6.984,148.985
C04498=1136.433,134.185,-57.841,-178.934,6.981,148.985
C04499=1136.438,133.935,-57.820,-178.937,6.980,148.986
C04500=1136.443,133.686,-57.800,-178.940,6.978,148.986
C04501=1136.447,133.437,-57.780,-178.942,6.976,148.987
C04502=1136.452,133.187,-57.760,-178.945,6.974,148.987
C04503=1136.456,132.938,-57.739,-178.948,6.972,148.987
C04504=1136.462,132.689,-57.720,-178.951,6.970,148.987
C04505=1136.466,132.440,-57.700,-178.953,6.968,148.988
C04506=1136.471,132.191,-57.680,-178.956,6.967,148.988
C04507=1136.476,131.942,-57.659,-178.959,6.965,148.989
C04508=1136.481,131.673,-57.638,-178.962,6.962,148.989
C04509=1136.486,131.405,-57.616,-178.965,6.961,148.990
C04510=1136.491,131.136,-57.595,-178.969,6.958,148.990
C04511=1136.497,130.867,-57.573,-178.971,6.957,148.990
C04512=1136.501,130.618,-57.553,-178.974,6.955,148.991
C04513=1136.507,130.369,-57.533,-178.977,6.953,148.991
C04514=1136.511,130.120,-57.513,-178.980,6.951,148.992
C04515=1136.516,129.871,-57.493,-178.983,6.949,148.992
C04516=1136.520,129.622,-57.473,-178.985,6.947,148.992
C04517=1136.525,129.373,-57.454,-178.988,6.945,148.993
C04518=1136.530,129.123,-57.434,-178.991,6.944,148.993
C04519=1136.535,128.874,-57.414,-178.993,6.942,148.993
C04520=1136.539,128.625,-57.394,-178.996,6.940,148.994
C04521=1136.544,128.377,-57.374,-178.999,6.938,148.994
C04522=1136.549,128.127,-57.354,-179.002,6.936,148.995
C04523=1136.554,127.877,-57.335,-179.005,6.935,148.995
C04524=1136.558,127.628,-57.314,-179.007,6.933,148.995
C04525=1136.564,127.380,-57.295,-179.010,6.931,148.996
C04526=1136.568,127.130,-57.275,-179.013,6.929,148.996
C04527=1136.573,126.881,-57.255,-179.016,6.928,148.997
C04528=1136.578,126.631,-57.235,-179.019,6.925,148.997
C04529=1136.583,126.383,-57.216,-179.022,6.924,148.997
C04530=1136.588,126.133,-57.196,-179.024,6.922,148.998
C04531=1136.592,125.884,-57.176,-179.027,6.920,148.998
C04532=1136.597,125.635,-57.157,-179.030,6.919,148.999
C04533=1136.602,125.386,-57.137,-179.033,6.917,148.999
C04534=1136.606,125.136,-57.118,-179.035,6.915,148.999
C04535=1136.611,124.887,-57.098,-179.039,6.913,149.000
C04536=1136.616,124.639,-57.078,-179.041,6.911,149.000
C04537=1136.621,124.389,-57.059,-179.044,6.909,149.001
C04538=1136.625,124.139,-57.039,-179.047,6.908,149.001
C04539=1136.631,123.891,-57.020,-179.050,6.906,149.001
C04540=1136.635,123.642,-56.999,-179.052,6.904,149.002
C04541=1136.640,123.392,-56.980,-179.055,6.903,149.002
C04542=1136.645,123.144,-56.961,-179.058,6.901,149.003
C04543=1136.649,122.894,-56.941,-179.060,6.899,149.003
C04544=1136.655,122.645,-56.922,-179.064,6.897,149.003
C04545=1136.659,122.395,-56.902,-179.067,6.895,149.004
C04546=1136.664,122.146,-56.883,-179.069,6.893,149.004
C04547=1136.669,121.897,-56.864,-179.072,6.892,149.005
C04548=1136.674,121.648,-56.844,-179.075,6.890,149.005
C04549=1136.678,121.398,-56.825,-179.077,6.888,149.005
C04550=1136.683,121.150,-56.805,-179.080,6.887,149.006
C04551=1136.688,120.900,-56.785,-179.083,6.885,149.006
C04552=1136.693,120.652,-56.766,-179.086,6.883,149.007
C04553=1136.697,120.402,-56.747,-179.088,6.881,149.007
C04554=1136.702,120.153,-56.727,-179.092,6.879,149.007
C04555=1136.708,119.904,-56.708,-179.094,6.877,149.008
C04556=1136.712,119.655,-56.689,-179.097,6.876,149.008
C04557=1136.717,119.406,-56.669,-179.100,6.874,149.009
C04558=1136.722,119.156,-56.650,-179.103,6.872,149.009
C04559=1136.727,118.907,-56.631,-179.105,6.871,149.009
C04560=1136.731,118.657,-56.612,-179.108,6.869,149.010
C04561=1136.736,118.408,-56.592,-179.111,6.867,149.010
C04562=1136.741,118.159,-56.573,-179.113,6.865,149.011
C04563=1136.745,117.910,-56.554,-179.116,6.864,149.011
C04564=1136.751,117.661,-56.535,-179.119,6.862,149.011
C04565=1136.755,117.411,-56.515,-179.122,6.860,149.012
C04566=1136.760,117.163,-56.496,-179.124,6.859,149.012
C04567=1136.765,116.913,-56.477,-179.127,6.857,149.013
C04568=1136.770,116.664,-56.458,-179.130,6.855,149.013
C04569=1136.774,116.414,-56.439,-179.133,6.853,149.013
C04570=1136.780,116.166,-56.420,-179.136,6.851,149.014
C04571=1136.785,115.916,-56.400,-179.139,6.850,149.014
C04572=1136.789,115.667,-56.381,-179.142,6.848,149.015
C04573=1136.794,115.417,-56.363,-179.145,6.847,149.015
C04574=1136.799,115.169,-56.344,-179.147,6.845,149.016
C04575=1136.804,114.919,-56.324,-179.150,6.843,149.016
C04576=1136.809,114.670,-56.305,-179.153,6.841,149.016
C04577=1136.813,114.420,-56.287,-179.156,6.840,149.017
C04578=1136.819,114.172,-56.267,-179.158,6.838,149.017
C04579=1136.823,113.922,-56.248,-179.161,6.836,149.018
C04580=1136.828,113.673,-56.229,-179.164,6.835,149.018
C04581=1136.833,113.423,-56.210,-179.166,6.833,149.019
C04582=1136.838,113.175,-56.191,-179.169,6.831,149.019
C04583=1136.843,112.926,-56.172,-179.172,6.830,149.019
C04584=1136.847,112.676,-56.154,-179.175,6.828,149.020
C04585=1136.853,112.427,-56.134,-179.177,6.826,149.020
C04586=1136.857,112.178,-56.115,-179.180,6.825,149.021
C04587=1136.862,111.928,-56.097,-179.183,6.823,149.021
C04588=1136.866,111.679,-56.078,-179.186,6.821,149.021
C04589=1136.872,111.430,-56.059,-179.189,6.820,149.022
C04590=1136.876,111.181,-56.040,-179.191,6.818,149.022
C04591=1136.881,110.931,-56.021,-179.194,6.817,149.023
C04592=1136.886,110.682,-56.003,-179.197,6.815,149.023
C04593=1136.891,110.433,-55.983,-179.200,6.813,149.024
C04594=1136.896,110.183,-55.965,-179.202,6.812,149.024
C04595=1136.901,109.935,-55.946,-179.205,6.810,149.024
C04596=1136.905,109.685,-55.927,-179.208,6.808,149.025
C04597=1136.910,109.436,-55.909,-179.211,6.807,149.025
C04598=1136.916,109.187,-55.890,-179.213,6.805,149.026
C04599=1136.920,108.937,-55.871,-179.216,6.803,149.026
C04600=1136.925,108.688,-55.853,-179.219,6.802,149.027
C04601=1136.930,108.439,-55.834,-179.222,6.800,149.027
C04602=1136.934,108.190,-55.816,-179.225,6.799,149.028
C04603=1136.940,107.941,-55.796,-179.227,6.797,149.028
C04604=1136.944,107.691,-55.778,-179.230,6.795,149.028
C04605=1136.949,107.442,-55.759,-179.233,6.794,149.029
C04606=1136.954,107.193,-55.741,-179.236,6.792,149.029
C04607=1136.958,106.943,-55.722,-179.238,6.790,149.030
C04608=1136.964,106.694,-55.703,-179.241,6.788,149.030
C04609=1136.969,106.445,-55.685,-179.244,6.787,149.030
C04610=1136.973,106.196,-55.666,-179.247,6.785,149.031
C04611=1136.978,105.946,-55.647,-179.249,6.783,149.031
C04612=1136.983,105.678,-55.628,-179.253,6.782,149.032
C04613=1136.988,105.410,-55.608,-179.256,6.780,149.032
C04614=1136.994,105.142,-55.588,-179.259,6.778,149.033
C04615=1136.999,104.873,-55.568,-179.261,6.776,149.033
C04616=1137.004,104.623,-55.549,-179.264,6.775,149.034
C04617=1137.009,104.375,-55.531,-179.267,6.773,149.034
C04618=1137.014,104.125,-55.513,-179.270,6.772,149.035
C04619=1137.018,103.876,-55.494,-179.273,6.770,149.035
C04620=1137.024,103.626,-55.476,-179.276,6.768,149.035
C04621=1137.028,103.378,-55.457,-179.278,6.767,149.036
C04622=1137.033,103.128,-55.439,-179.281,6.765,149.036
C04623=1137.037,102.878,-55.421,-179.284,6.763,149.037
C04624=1137.043,102.629,-55.402,-179.286,6.762,149.037
C04625=1137.048,102.380,-55.384,-179.289,6.760,149.037
C04626=1137.053,102.131,-55.366,-179.292,6.759,149.038
C04627=1137.057,101.881,-55.347,-179.295,6.758,149.039
C04628=1137.062,101.632,-55.329,-179.297,6.756,149.039
C04629=1137.068,101.383,-55.311,-179.300,6.754,149.039
C04630=1137.072,101.134,-55.293,-179.303,6.753,149.040
C04631=1137.077,100.885,-55.274,-179.306,6.751,149.040
C04632=1137.081,100.635,-55.256,-179.308,6.749,149.041
C04633=1137.086,100.386,-55.238,-179.311,6.748,149.041
C04634=1137.092,100.136,-55.219,-179.314,6.746,149.042
C04635=1137.097,99.887,-55.201,-179.317,6.745,149.042
C04636=1137.102,99.638,-55.183,-179.320,6.743,149.042
C04637=1137.106,99.388,-55.165,-179.322,6.741,149.043
C04638=1137.111,99.139,-55.147,-179.325,6.740,149.043
C04639=1137.116,98.890,-55.129,-179.328,6.738,149.044
C04640=1137.121,98.641,-55.111,-179.331,6.736,149.044
C04641=1137.126,98.392,-55.093,-179.333,6.736,149.045
C04642=1137.131,98.142,-55.075,-179.336,6.734,149.045
C04643=1137.135,97.892,-55.057,-179.339,6.733,149.046
C04644=1137.141,97.643,-55.038,-179.341,6.731,149.046
C04645=1137.145,97.394,-55.020,-179.344,6.729,149.046
C04646=1137.150,97.145,-55.002,-179.347,6.728,149.047
C04647=1137.155,96.895,-54.984,-179.350,6.726,149.047
C04648=1137.160,96.646,-54.966,-179.353,6.725,149.048
C04649=1137.165,96.397,-54.948,-179.356,6.723,149.048
C04650=1137.170,96.148,-54.930,-179.358,6.721,149.049
C04651=1137.174,95.898,-54.912,-179.360,6.720,149.049
C04652=1137.179,95.649,-54.894,-179.363,6.719,149.050
C04653=1137.184,95.400,-54.876,-179.366,6.717,149.050
C04654=1137.189,95.151,-54.858,-179.369,6.715,149.050
C04655=1137.194,94.901,-54.840,-179.372,6.714,149.051
C04656=1137.199,94.652,-54.822,-179.375,6.712,149.052
C04657=1137.204,94.403,-54.804,-179.377,6.711,149.052
C04658=1137.209,94.153,-54.787,-179.380,6.709,149.052
C04659=1137.214,93.904,-54.769,-179.383,6.707,149.053
C04660=1137.219,93.655,-54.751,-179.385,6.707,149.053
C04661=1137.224,93.406,-54.733,-179.388,6.705,149.054
C04662=1137.229,93.157,-54.715,-179.391,6.704,149.054
C04663=1137.234,92.907,-54.697,-179.394,6.702,149.055
C04664=1137.238,92.657,-54.679,-179.396,6.700,149.055
C04665=1137.242,92.408,-54.662,-179.399,6.699,149.056
C04666=1137.247,92.159,-54.644,-179.402,6.697,149.056
C04667=1137.252,91.910,-54.626,-179.405,6.695,149.056
C04668=1137.257,91.660,-54.609,-179.407,6.695,149.057
C04669=1137.262,91.411,-54.591,-179.410,6.693,149.057
C04670=1137.267,91.161,-54.573,-179.413,6.691,149.058
C04671=1137.272,90.912,-54.555,-179.416,6.690,149.058
C04672=1137.277,90.662,-54.537,-179.418,6.688,149.059
C04673=1137.282,90.413,-54.519,-179.421,6.686,149.059
C04674=1137.286,90.164,-54.502,-179.424,6.685,149.060
C04675=1137.292,89.915,-54.485,-179.426,6.684,149.060
C04676=1137.297,89.665,-54.467,-179.429,6.683,149.061
C04677=1137.302,89.416,-54.449,-179.432,6.681,149.061
C04678=1137.307,89.167,-54.431,-179.435,6.679,149.061
C04679=1137.312,88.917,-54.413,-179.438,6.678,149.062
C04680=1137.316,88.668,-54.397,-179.441,6.676,149.063
C04681=1137.321,88.419,-54.379,-179.443,6.675,149.063
C04682=1137.326,88.169,-54.361,-179.445,6.674,149.063
C04683=1137.331,87.920,-54.344,-179.448,6.672,149.064
C04684=1137.337,87.671,-54.326,-179.451,6.670,149.064
C04685=1137.341,87.422,-54.309,-179.454,6.669,149.065
C04686=1137.346,87.173,-54.291,-179.457,6.667,149.065
C04687=1137.351,86.923,-54.274,-179.459,6.667,149.066
C04688=1137.356,86.674,-54.256,-179.462,6.665,149.066
C04689=1137.360,86.425,-54.239,-179.465,6.663,149.067
C04690=1137.366,86.175,-54.221,-179.468,6.662,149.067
C04691=1137.371,85.926,-54.203,-179.470,6.660,149.068
C04692=1137.376,85.676,-54.186,-179.473,6.659,149.068
C04693=1137.380,85.427,-54.169,-179.475,6.658,149.068
C04694=1137.385,85.177,-54.152,-179.478,6.656,149.069
C04695=1137.390,84.928,-54.134,-179.481,6.655,149.070
C04696=1137.395,84.679,-54.117,-179.484,6.653,149.070
C04697=1137.400,84.430,-54.100,-179.487,6.652,149.070
C04698=1137.405,84.180,-54.082,-179.489,6.651,149.071
C04699=1137.410,83.931,-54.065,-179.492,6.649,149.071
C04700=1137.415,83.682,-54.047,-179.495,6.648,149.072
C04701=1137.420,83.432,-54.030,-179.498,6.646,149.072
C04702=1137.424,83.182,-54.013,-179.500,6.644,149.073
C04703=1137.429,82.933,-53.995,-179.503,6.644,149.073
C04704=1137.434,82.683,-53.978,-179.505,6.642,149.074
C04705=1137.440,82.435,-53.962,-179.509,6.641,149.074
C04706=1137.444,82.186,-53.944,-179.511,6.639,149.075
C04707=1137.449,81.936,-53.927,-179.514,6.637,149.075
C04708=1137.454,81.686,-53.910,-179.516,6.636,149.076
C04709=1137.459,81.437,-53.892,-179.519,6.635,149.076
C04710=1137.464,81.188,-53.875,-179.522,6.633,149.077
C04711=1137.469,80.938,-53.858,-179.525,6.632,149.077
C04712=1137.474,80.690,-53.841,-179.528,6.630,149.077
C04713=1137.479,80.440,-53.824,-179.530,6.629,149.078
C04714=1137.484,80.190,-53.806,-179.533,6.628,149.079
C04715=1137.488,79.941,-53.790,-179.536,6.626,149.079
C04716=1137.494,79.673,-53.771,-179.539,6.625,149.079
C04717=1137.499,79.404,-53.753,-179.542,6.623,149.080
C04718=1137.505,79.136,-53.734,-179.544,6.622,149.081
C04719=1137.510,78.867,-53.716,-179.547,6.620,149.081
C04720=1137.515,78.618,-53.699,-179.550,6.619,149.082
C04721=1137.520,78.368,-53.682,-179.553,6.618,149.082
C04722=1137.525,78.119,-53.665,-179.555,6.616,149.082
C04723=1137.530,77.870,-53.647,-179.558,6.615,149.083
C04724=1137.534,77.621,-53.631,-179.561,6.613,149.083
C04725=1137.540,77.371,-53.614,-179.563,6.613,149.084
C04726=1137.545,77.122,-53.597,-179.566,6.611,149.084
C04727=1137.550,76.872,-53.580,-179.569,6.609,149.085
C04728=1137.554,76.623,-53.563,-179.572,6.608,149.085
C04729=1137.560,76.373,-53.546,-179.574,6.607,149.086
C04730=1137.565,76.124,-53.530,-179.577,6.605,149.086
C04731=1137.569,75.875,-53.513,-179.580,6.604,149.087
C04732=1137.574,75.626,-53.495,-179.583,6.602,149.087
C04733=1137.579,75.376,-53.478,-179.585,6.602,149.088
C04734=1137.584,75.127,-53.461,-179.588,6.600,149.088
C04735=1137.589,74.878,-53.445,-179.591,6.598,149.089
C04736=1137.593,74.628,-53.428,-179.593,6.597,149.089
C04737=1137.599,74.379,-53.411,-179.596,6.596,149.090
C04738=1137.604,74.129,-53.395,-179.599,6.595,149.090
C04739=1137.609,73.880,-53.377,-179.602,6.593,149.091
C04740=1137.614,73.631,-53.361,-179.604,6.591,149.091
C04741=1137.618,73.381,-53.344,-179.606,6.590,149.092
C04742=1137.624,73.132,-53.327,-179.610,6.589,149.092
C04743=1137.629,72.883,-53.311,-179.612,6.587,149.093
C04744=1137.633,72.633,-53.294,-179.615,6.587,149.093
C04745=1137.638,72.384,-53.277,-179.617,6.585,149.093
C04746=1137.644,72.134,-53.261,-179.621,6.584,149.094
C04747=1137.648,71.885,-53.245,-179.623,6.582,149.095
C04748=1137.653,71.635,-53.227,-179.625,6.581,149.095
C04749=1137.659,71.386,-53.211,-179.628,6.579,149.095
C04750=1137.663,71.137,-53.194,-179.631,6.578,149.096
C04751=1137.668,70.887,-53.177,-179.634,6.577,149.097
C04752=1137.673,70.638,-53.161,-179.636,6.576,149.097
C04753=1137.678,70.389,-53.144,-179.639,6.574,149.097
C04754=1137.683,70.139,-53.127,-179.642,6.573,149.098
C04755=1137.688,69.889,-53.111,-179.645,6.572,149.098
C04756=1137.693,69.640,-53.095,-179.647,6.570,149.099
C04757=1137.698,69.391,-53.078,-179.650,6.569,149.099
C04758=1137.703,69.141,-53.061,-179.653,6.568,149.100
C04759=1137.708,68.892,-53.044,-179.655,6.566,149.100
C04760=1137.713,68.642,-53.029,-179.658,6.565,149.101
C04761=1137.718,68.393,-53.012,-179.661,6.564,149.102
C04762=1137.723,68.144,-52.995,-179.664,6.563,149.102
C04763=1137.728,67.894,-52.979,-179.666,6.561,149.102
C04764=1137.733,67.645,-52.963,-179.668,6.560,149.103
C04765=1137.738,67.395,-52.946,-179.672,6.559,149.104
C04766=1137.742,67.146,-52.930,-179.674,6.557,149.104
C04767=1137.748,66.897,-52.913,-179.677,6.556,149.104
C04768=1137.753,66.647,-52.897,-179.679,6.555,149.105
C04769=1137.758,66.398,-52.880,-179.683,6.554,149.105
C04770=1137.762,66.148,-52.864,-179.685,6.553,149.106
C04771=1137.768,65.899,-52.848,-179.687,6.551,149.106
C04772=1137.772,65.650,-52.832,-179.690,6.549,149.107
C04773=1137.777,65.401,-52.815,-179.693,6.549,149.107
C04774=1137.783,65.150,-52.799,-179.696,6.547,149.108
C04775=1137.787,64.901,-52.782,-179.698,6.546,149.108
C04776=1137.792,64.652,-52.766,-179.701,6.545,149.109
C04777=1137.797,64.402,-52.750,-179.704,6.543,149.109
C04778=1137.802,64.153,-52.733,-179.706,6.542,149.110
C04779=1137.807,63.903,-52.717,-179.709,6.541,149.110
C04780=1137.812,63.654,-52.701,-179.712,6.540,149.111
C04781=1137.817,63.405,-52.685,-179.715,6.538,149.111
C04782=1137.822,63.155,-52.669,-179.717,6.537,149.112
C04783=1137.826,62.906,-52.652,-179.720,6.536,149.112
C04784=1137.833,62.656,-52.636,-179.723,6.534,149.113
C04785=1137.837,62.407,-52.619,-179.725,6.533,149.113
C04786=1137.842,62.157,-52.604,-179.728,6.532,149.114
C04787=1137.847,61.908,-52.587,-179.731,6.531,149.114
C04788=1137.852,61.658,-52.572,-179.733,6.530,149.115
C04789=1137.857,61.410,-52.555,-179.736,6.528,149.115
C04790=1137.862,61.160,-52.539,-179.739,6.526,149.116
C04791=1137.867,60.911,-52.523,-179.741,6.526,149.116
C04792=1137.872,60.661,-52.507,-179.744,6.524,149.117
C04793=1137.877,60.412,-52.491,-179.746,6.523,149.117
C04794=1137.882,60.162,-52.475,-179.749,6.522,149.118
C04795=1137.887,59.913,-52.458,-179.752,6.521,149.118
C04796=1137.892,59.663,-52.443,-179.754,6.520,149.119
C04797=1137.897,59.414,-52.427,-179.757,6.518,149.119
C04798=1137.902,59.165,-52.411,-179.760,6.517,149.120
C04799=1137.907,58.915,-52.395,-179.762,6.516,149.120
C04800=1137.912,58.666,-52.378,-179.765,6.514,149.121
C04801=1137.917,58.416,-52.362,-179.768,6.514,149.122
C04802=1137.922,58.166,-52.347,-179.771,6.512,149.122
C04803=1137.927,57.918,-52.331,-179.773,6.511,149.122
C04804=1137.931,57.668,-52.315,-179.776,6.510,149.123
C04805=1137.937,57.418,-52.300,-179.779,6.508,149.123
C04806=1137.941,57.169,-52.283,-179.781,6.508,149.124
C04807=1137.947,56.920,-52.267,-179.784,6.506,149.124
C04808=1137.952,56.670,-52.252,-179.787,6.505,149.125
C04809=1137.957,56.421,-52.235,-179.789,6.504,149.125
C04810=1137.962,56.171,-52.219,-179.792,6.502,149.126
C04811=1137.967,55.922,-52.204,-179.794,6.502,149.127
C04812=1137.972,55.672,-52.188,-179.797,6.500,149.127
C04813=1137.977,55.423,-52.172,-179.800,6.498,149.127
C04814=1137.982,55.174,-52.157,-179.802,6.498,149.128
C04815=1137.987,54.924,-52.141,-179.805,6.496,149.129
C04816=1137.992,54.674,-52.125,-179.807,6.495,149.129
C04817=1137.997,54.426,-52.109,-179.810,6.494,149.129
C04818=1138.002,54.175,-52.093,-179.813,6.493,149.130
C04819=1138.007,53.926,-52.077,-179.816,6.492,149.131
C04820=1138.013,53.658,-52.060,-179.818,6.490,149.131
C04821=1138.018,53.389,-52.044,-179.822,6.489,149.132
C04822=1138.023,53.120,-52.026,-179.824,6.487,149.132
C04823=1138.028,52.852,-52.009,-179.827,6.487,149.133
C04824=1138.034,52.602,-51.994,-179.830,6.485,149.133
C04825=1138.039,52.353,-51.978,-179.832,6.485,149.134
C04826=1138.044,52.103,-51.962,-179.835,6.483,149.134
C04827=1138.048,51.854,-51.947,-179.838,6.481,149.135
C04828=1138.054,51.604,-51.932,-179.840,6.481,149.135
C04829=1138.059,51.355,-51.916,-179.843,6.479,149.136
C04830=1138.064,51.105,-51.900,-179.845,6.478,149.136
C04831=1138.069,50.856,-51.885,-179.848,6.477,149.137
C04832=1138.074,50.606,-51.870,-179.851,6.476,149.137
C04833=1138.079,50.358,-51.853,-179.854,6.475,149.138
C04834=1138.083,50.108,-51.838,-179.856,6.474,149.138
C04835=1138.088,49.858,-51.822,-179.859,6.473,149.139
C04836=1138.094,49.609,-51.807,-179.862,6.471,149.139
C04837=1138.099,49.360,-51.791,-179.864,6.470,149.140
C04838=1138.103,49.110,-51.776,-179.867,6.469,149.141
C04839=1138.109,48.860,-51.760,-179.869,6.468,149.141
C04840=1138.114,48.611,-51.745,-179.872,6.466,149.141
C04841=1138.119,48.362,-51.730,-179.875,6.466,149.142
C04842=1138.123,48.112,-51.714,-179.877,6.464,149.143
C04843=1138.129,47.862,-51.698,-179.880,6.463,149.143
C04844=1138.134,47.613,-51.683,-179.883,6.462,149.144
C04845=1138.139,47.363,-51.668,-179.885,6.461,149.144
C04846=1138.145,47.114,-51.653,-179.888,6.460,149.145
C04847=1138.149,46.864,-51.637,-179.891,6.458,149.145
C04848=1138.154,46.615,-51.622,-179.893,6.458,149.146
C04849=1138.159,46.366,-51.607,-179.896,6.456,149.146
C04850=1138.164,46.116,-51.591,-179.898,6.455,149.147
C04851=1138.169,45.867,-51.576,-179.901,6.454,149.147
C04852=1138.174,45.617,-51.560,-179.904,6.453,149.148
C04853=1138.179,45.368,-51.545,-179.906,6.451,149.148
C04854=1138.184,45.118,-51.530,-179.909,6.451,149.149
C04855=1138.189,44.868,-51.515,-179.912,6.449,149.149
C04856=1138.195,44.619,-51.499,-179.914,6.449,149.150
C04857=1138.199,44.370,-51.484,-179.917,6.447,149.150
C04858=1138.204,44.120,-51.468,-179.919,6.446,149.151
C04859=1138.209,43.871,-51.453,-179.922,6.445,149.151
C04860=1138.214,43.621,-51.438,-179.925,6.444,149.152
C04861=1138.219,43.372,-51.423,-179.927,6.443,149.152
C04862=1138.224,43.122,-51.408,-179.930,6.442,149.153
C04863=1138.229,42.873,-51.393,-179.933,6.441,149.154
C04864=1138.235,42.623,-51.378,-179.935,6.440,149.154
C04865=1138.239,42.374,-51.363,-179.938,6.438,149.154
C04866=1138.244,42.124,-51.347,-179.940,6.438,149.155
C04867=1138.250,41.875,-51.331,-179.943,6.436,149.156
C04868=1138.255,41.625,-51.317,-179.945,6.435,149.156
C04869=1138.259,41.376,-51.302,-179.949,6.434,149.157
C04870=1138.265,41.126,-51.286,-179.951,6.433,149.157
C04871=1138.269,40.877,-51.271,-179.953,6.432,149.158
C04872=1138.275,40.627,-51.257,-179.956,6.431,149.158
C04873=1138.280,40.378,-51.242,-179.959,6.429,149.159
C04874=1138.285,40.129,-51.226,-179.961,6.429,149.159
C04875=1138.290,39.879,-51.212,-179.964,6.427,149.160
C04876=1138.295,39.630,-51.196,-179.966,6.427,149.160
C04877=1138.300,39.380,-51.182,-179.969,6.425,149.161
C04878=1138.305,39.130,-51.166,-179.972,6.424,149.161
C04879=1138.310,38.881,-51.151,-179.975,6.423,149.162
C04880=1138.315,38.631,-51.137,-179.977,6.422,149.162
C04881=1138.320,38.382,-51.121,-179.980,6.421,149.163
C04882=1138.325,38.132,-51.107,-179.982,6.420,149.163
C04883=1138.330,37.882,-51.091,-179.985,6.419,149.164
C04884=1138.335,37.633,-51.076,-179.988,6.418,149.165
C04885=1138.340,37.384,-51.062,-179.990,6.417,149.165
C04886=1138.345,37.134,-51.046,-179.993,6.416,149.166
C04887=1138.350,36.885,-51.032,-179.995,6.415,149.166
C04888=1138.356,36.635,-51.017,-179.998,6.413,149.167
C04889=1138.361,36.385,-51.002,179.999,6.413,149.167
C04890=1138.365,36.136,-50.987,179.997,6.411,149.168
C04891=1138.371,35.886,-50.972,179.994,6.410,149.168
C04892=1138.376,35.637,-50.957,179.991,6.409,149.169
C04893=1138.381,35.388,-50.943,179.989,6.408,149.169
C04894=1138.386,35.138,-50.928,179.987,6.407,149.170
C04895=1138.391,34.888,-50.913,179.984,6.406,149.170
C04896=1138.396,34.639,-50.898,179.982,6.405,149.171
C04897=1138.401,34.389,-50.883,179.979,6.404,149.171
C04898=1138.406,34.140,-50.868,179.976,6.403,149.172
C04899=1138.411,33.890,-50.854,179.973,6.402,149.172
C04900=1138.417,33.640,-50.839,179.971,6.401,149.173
C04901=1138.421,33.391,-50.824,179.968,6.400,149.174
C04902=1138.427,33.142,-50.810,179.966,6.399,149.174
C04903=1138.431,32.893,-50.795,179.964,6.398,149.174
C04904=1138.437,32.643,-50.780,179.960,6.397,149.175
C04905=1138.442,32.394,-50.766,179.958,6.396,149.176
C04906=1138.447,32.144,-50.751,179.955,6.394,149.176
C04907=1138.452,31.895,-50.737,179.953,6.394,149.177
C04908=1138.457,31.645,-50.722,179.950,6.392,149.177
C04909=1138.462,31.396,-50.707,179.947,6.392,149.178
C04910=1138.467,31.146,-50.693,179.945,6.391,149.178
C04911=1138.472,30.896,-50.678,179.942,6.389,149.179
C04912=1138.477,30.647,-50.663,179.940,6.389,149.179
C04913=1138.482,30.397,-50.649,179.937,6.387,149.180
C04914=1138.487,30.147,-50.634,179.935,6.386,149.180
C04915=1138.493,29.898,-50.620,179.932,6.386,149.181
C04916=1138.497,29.649,-50.605,179.929,6.384,149.181
C04917=1138.502,29.400,-50.591,179.927,6.383,149.182
C04918=1138.507,29.150,-50.577,179.924,6.382,149.183
C04919=1138.513,28.900,-50.562,179.922,6.381,149.183
C04920=1138.518,28.651,-50.547,179.919,6.380,149.183
C04921=1138.523,28.401,-50.533,179.916,6.379,149.184
C04922=1138.528,28.151,-50.518,179.914,6.379,149.185
C04923=1138.533,27.902,-50.505,179.911,6.377,149.185
C04924=1138.538,27.634,-50.489,179.909,6.376,149.186
C04925=1138.544,27.364,-50.473,179.906,6.375,149.186
C04926=1138.550,27.095,-50.458,179.903,6.374,149.187
C04927=1138.555,26.826,-50.442,179.900,6.373,149.188
C04928=1138.560,26.577,-50.428,179.898,6.372,149.188
C04929=1138.565,26.327,-50.413,179.895,6.371,149.188
C04930=1138.570,26.078,-50.399,179.893,6.370,149.189
C04931=1138.576,25.828,-50.384,179.890,6.369,149.190
C04932=1138.581,25.579,-50.370,179.888,6.368,149.190
C04933=1138.585,25.329,-50.355,179.885,6.367,149.191
C04934=1138.590,25.079,-50.341,179.882,6.366,149.191
C04935=1138.595,24.830,-50.327,179.880,6.365,149.192
C04936=1138.601,24.581,-50.313,179.877,6.365,149.192
C04937=1138.606,24.331,-50.298,179.875,6.363,149.193
C04938=1138.611,24.081,-50.284,179.872,6.362,149.193
C04939=1138.616,23.831,-50.270,179.869,6.361,149.194
C04940=1138.621,23.582,-50.256,179.867,6.360,149.194
C04941=1138.626,23.333,-50.242,179.864,6.360,149.195
C04942=1138.631,23.083,-50.227,179.862,6.358,149.196
C04943=1138.636,22.833,-50.213,179.859,6.357,149.196
C04944=1138.641,22.584,-50.199,179.857,6.357,149.197
C04945=1138.647,22.335,-50.185,179.854,6.355,149.197
C04946=1138.652,22.085,-50.171,179.851,6.355,149.198
C04947=1138.657,21.835,-50.156,179.849,6.354,149.198
C04948=1138.662,21.585,-50.142,179.846,6.352,149.199
C04949=1138.667,21.336,-50.128,179.844,6.352,149.199
C04950=1138.672,21.087,-50.114,179.841,6.350,149.200
C04951=1138.677,20.837,-50.100,179.839,6.349,149.200
C04952=1138.682,20.587,-50.085,179.836,6.349,149.201
C04953=1138.688,20.338,-50.072,179.833,6.347,149.201
C04954=1138.693,20.089,-50.057,179.831,6.347,149.202
C04955=1138.697,19.839,-50.043,179.829,6.346,149.203
C04956=1138.702,19.589,-50.029,179.826,6.344,149.203
C04957=1138.707,19.340,-50.015,179.823,6.344,149.204
C04958=1138.713,19.090,-50.002,179.821,6.343,149.204
C04959=1138.717,18.840,-49.988,179.818,6.342,149.205
C04960=1138.723,18.591,-49.974,179.816,6.341,149.205
C04961=1138.728,18.342,-49.959,179.813,6.340,149.206
C04962=1138.733,18.092,-49.945,179.811,6.339,149.206
C04963=1138.739,17.843,-49.931,179.808,6.338,149.207
C04964=1138.744,17.593,-49.918,179.806,6.337,149.207
C04965=1138.748,17.343,-49.904,179.803,6.336,149.208
C04966=1138.753,17.094,-49.890,179.800,6.335,149.209
C04967=1138.758,16.845,-49.876,179.798,6.335,149.209
C04968=1138.763,16.595,-49.861,179.795,6.333,149.210
C04969=1138.769,16.344,-49.848,179.793,6.332,149.210
C04970=1138.774,16.095,-49.834,179.791,6.332,149.211
C04971=1138.778,15.846,-49.820,179.788,6.331,149.211
C04972=1138.784,15.597,-49.806,179.785,6.330,149.212
C04973=1138.789,15.347,-49.792,179.783,6.329,149.212
C04974=1138.794,15.097,-49.779,179.780,6.328,149.213
C04975=1138.800,14.848,-49.765,179.778,6.327,149.213
C04976=1138.805,14.598,-49.750,179.775,6.326,149.214
C04977=1138.809,14.348,-49.737,179.773,6.325,149.214
C04978=1138.815,14.099,-49.723,179.770,6.324,149.215
C04979=1138.820,13.850,-49.709,179.767,6.323,149.216
C04980=1138.825,13.599,-49.696,179.765,6.323,149.216
C04981=1138.830,13.351,-49.682,179.762,6.321,149.217
C04982=1138.835,13.101,-49.668,179.760,6.321,149.217
C04983=1138.841,12.851,-49.655,179.758,6.320,149.218
C04984=1138.846,12.601,-49.641,179.755,6.319,149.218
C04985=1138.850,12.352,-49.627,179.752,6.318,149.219
C04986=1138.856,12.102,-49.614,179.750,6.317,149.219
C04987=1138.861,11.853,-49.599,179.747,6.316,149.220
C04988=1138.866,11.604,-49.586,179.745,6.315,149.220
C04989=1138.871,11.354,-49.573,179.742,6.314,149.221
C04990=1138.876,11.105,-49.559,179.740,6.314,149.222
C04991=1138.882,10.854,-49.545,179.738,6.313,149.222
C04992=1138.886,10.605,-49.531,179.734,6.312,149.223
C04993=1138.891,10.356,-49.517,179.732,6.311,149.223
C04994=1138.897,10.106,-49.504,179.730,6.310,149.224
C04995=1138.901,9.857,-49.491,179.727,6.309,149.224
C04996=1138.907,9.607,-49.477,179.725,6.308,149.225
C04997=1138.912,9.358,-49.463,179.722,6.307,149.225
C04998=1138.917,9.108,-49.450,179.720,6.307,149.226
C04999=1138.922,8.859,-49.436,179.717,6.305,149.226
C05000=1138.928,8.608,-49.423,179.714,6.305,149.227
C05001=1138.932,8.359,-49.409,179.712,6.304,149.228
C05002=1138.938,8.109,-49.396,179.710,6.303,149.228
C05003=1138.943,7.859,-49.382,179.707,6.302,149.229
C05004=1138.948,7.610,-49.369,179.705,6.301,149.229
C05005=1138.953,7.360,-49.355,179.702,6.301,149.230
C05006=1138.958,7.111,-49.342,179.700,6.300,149.230
C05007=1138.963,6.861,-49.328,179.697,6.298,149.231
C05008=1138.969,6.612,-49.315,179.694,6.298,149.231
C05009=1138.973,6.362,-49.302,179.692,6.297,149.232
C05010=1138.979,6.113,-49.288,179.690,6.296,149.232
C05011=1138.983,5.863,-49.275,179.687,6.295,149.233
C05012=1138.989,5.614,-49.261,179.685,6.294,149.234
C05013=1138.994,5.363,-49.247,179.682,6.294,149.234
C05014=1138.999,5.114,-49.235,179.680,6.293,149.235
C05015=1139.005,4.865,-49.221,179.677,6.291,149.235
C05016=1139.009,4.615,-49.208,179.674,6.291,149.236
C05017=1139.015,4.365,-49.195,179.672,6.290,149.236
C05018=1139.019,4.116,-49.181,179.670,6.289,149.237
C05019=1139.025,3.866,-49.168,179.667,6.288,149.237
C05020=1139.030,3.616,-49.155,179.665,6.287,149.238
C05021=1139.035,3.367,-49.141,179.662,6.287,149.239
C05022=1139.040,3.117,-49.128,179.660,6.286,149.239
C05023=1139.046,2.868,-49.115,179.658,6.285,149.240
C05024=1139.050,2.618,-49.101,179.654,6.284,149.240
C05025=1139.056,2.369,-49.088,179.652,6.283,149.241
C05026=1139.061,2.119,-49.075,179.650,6.282,149.241
C05027=1139.066,1.869,-49.062,179.647,6.282,149.242
C05028=1139.071,1.600,-49.047,179.644,6.280,149.242
C05029=1139.077,1.331,-49.033,179.642,6.280,149.243
C05030=1139.083,1.061,-49.018,179.639,6.279,149.244
C05031=1139.088,0.791,-49.005,179.636,6.278,149.244
C05032=1139.093,0.542,-48.991,179.634,6.277,149.245
C05033=1139.099,0.293,-48.979,179.632,6.277,149.245
C05034=1139.104,0.043,-48.965,179.629,6.275,149.246
C05035=1139.109,-0.206,-48.952,179.626,6.275,149.246
C05036=1139.114,-0.457,-48.938,179.624,6.274,149.247
C05037=1139.119,-0.706,-48.926,179.622,6.273,149.247
C05038=1139.124,-0.955,-48.913,179.619,6.272,149.248
C05039=1139.129,-1.205,-48.899,179.616,6.271,149.249
C05040=1139.134,-1.454,-48.886,179.614,6.270,149.249
C05041=1139.140,-1.704,-48.873,179.611,6.270,149.250
C05042=1139.145,-1.954,-48.860,179.609,6.269,149.250
C05043=1139.150,-2.203,-48.848,179.607,6.268,149.251
C05044=1139.155,-2.454,-48.834,179.604,6.267,149.251
C05045=1139.160,-2.703,-48.821,179.602,6.266,149.252
C05046=1139.165,-2.952,-48.809,179.599,6.266,149.252
C05047=1139.170,-3.202,-48.795,179.597,6.265,149.253
C05048=1139.175,-3.451,-48.782,179.594,6.264,149.254
C05049=1139.180,-3.701,-48.769,179.591,6.263,149.254
C05050=1139.186,-3.951,-48.756,179.589,6.262,149.255
C05051=1139.191,-4.200,-48.743,179.587,6.262,149.255
C05052=1139.196,-4.450,-48.731,179.584,6.261,149.256
C05053=1139.202,-4.699,-48.717,179.582,6.260,149.256
C05054=1139.206,-4.949,-48.704,179.580,6.260,149.257
C05055=1139.211,-5.199,-48.692,179.577,6.258,149.257
C05056=1139.217,-5.448,-48.679,179.574,6.258,149.258
C05057=1139.222,-5.698,-48.666,179.572,6.257,149.258
C05058=1139.227,-5.948,-48.653,179.570,6.256,149.259
C05059=1139.233,-6.197,-48.640,179.567,6.255,149.260
C05060=1139.237,-6.447,-48.627,179.565,6.255,149.260
C05061=1139.242,-6.697,-48.614,179.562,6.253,149.261
C05062=1139.248,-6.946,-48.602,179.560,6.253,149.261
C05063=1139.253,-7.196,-48.588,179.557,6.252,149.262
C05064=1139.258,-7.446,-48.576,179.555,6.251,149.262
C05065=1139.263,-7.695,-48.563,179.553,6.251,149.263
C05066=1139.268,-7.944,-48.550,179.550,6.250,149.263
C05067=1139.274,-8.194,-48.537,179.547,6.249,149.264
C05068=1139.279,-8.444,-48.525,179.545,6.248,149.265
C05069=1139.284,-8.694,-48.512,179.543,6.247,149.265
C05070=1139.289,-8.943,-48.500,179.540,6.247,149.266
C05071=1139.294,-9.192,-48.487,179.538,6.246,149.266
C05072=1139.300,-9.443,-48.473,179.535,6.245,149.267
C05073=1139.305,-9.692,-48.461,179.533,6.245,149.267
C05074=1139.310,-9.941,-48.448,179.530,6.243,149.268
C05075=1139.315,-10.191,-48.436,179.528,6.243,149.268
C05076=1139.319,-10.441,-48.423,179.525,6.242,149.269
C05077=1139.326,-10.691,-48.410,179.523,6.241,149.269
C05078=1139.331,-10.940,-48.398,179.521,6.241,149.270
C05079=1139.336,-11.190,-48.385,179.518,6.240,149.271
C05080=1139.341,-11.439,-48.372,179.516,6.239,149.271
C05081=1139.346,-11.689,-48.359,179.513,6.238,149.272
C05082=1139.351,-11.939,-48.348,179.511,6.237,149.272
C05083=1139.356,-12.188,-48.335,179.508,6.237,149.273
C05084=1139.362,-12.438,-48.322,179.506,6.236,149.273
C05085=1139.367,-12.687,-48.309,179.504,6.235,149.274
C05086=1139.372,-12.937,-48.296,179.501,6.235,149.275
C05087=1139.377,-13.187,-48.284,179.499,6.234,149.275
C05088=1139.382,-13.436,-48.272,179.496,6.233,149.276
C05089=1139.387,-13.686,-48.259,179.493,6.232,149.276
C05090=1139.393,-13.936,-48.247,179.491,6.231,149.277
C05091=1139.397,-14.186,-48.234,179.489,6.231,149.277
C05092=1139.402,-14.435,-48.222,179.486,6.230,149.278
C05093=1139.407,-14.684,-48.209,179.484,6.229,149.278
C05094=1139.414,-14.935,-48.197,179.482,6.229,149.279
C05095=1139.419,-15.184,-48.184,179.479,6.228,149.279
C05096=1139.424,-15.433,-48.171,179.477,6.227,149.280
C05097=1139.429,-15.683,-48.160,179.475,6.227,149.281
C05098=1139.434,-15.933,-48.147,179.472,6.225,149.281
C05099=1139.439,-16.182,-48.134,179.469,6.225,149.282
C05100=1139.444,-16.432,-48.122,179.467,6.224,149.282
C05101=1139.450,-16.682,-48.109,179.465,6.223,149.283
C05102=1139.455,-16.931,-48.097,179.462,6.222,149.283
C05103=1139.460,-17.181,-48.085,179.460,6.222,149.284
C05104=1139.465,-17.430,-48.072,179.457,6.221,149.285
C05105=1139.471,-17.680,-48.061,179.455,6.220,149.285
C05106=1139.476,-17.930,-48.048,179.453,6.220,149.285
C05107=1139.480,-18.180,-48.035,179.450,6.219,149.286
C05108=1139.486,-18.430,-48.023,179.447,6.218,149.287
C05109=1139.491,-18.679,-48.010,179.445,6.217,149.287
C05110=1139.496,-18.929,-47.999,179.443,6.216,149.288
C05111=1139.501,-19.178,-47.986,179.440,6.216,149.288
C05112=1139.507,-19.428,-47.974,179.438,6.215,149.289
C05113=1139.512,-19.677,-47.961,179.436,6.214,149.289
C05114=1139.517,-19.927,-47.950,179.433,6.214,149.290
C05115=1139.522,-20.177,-47.937,179.431,6.213,149.291
C05116=1139.528,-20.427,-47.925,179.429,6.212,149.291
C05117=1139.533,-20.676,-47.913,179.426,6.212,149.292
C05118=1139.538,-20.926,-47.901,179.424,6.211,149.292
C05119=1139.543,-21.175,-47.889,179.422,6.210,149.293
C05120=1139.548,-21.425,-47.877,179.419,6.209,149.293
C05121=1139.553,-21.674,-47.864,179.416,6.209,149.294
C05122=1139.558,-21.925,-47.852,179.414,6.208,149.294
C05123=1139.563,-22.174,-47.839,179.411,6.207,149.295
C05124=1139.569,-22.424,-47.827,179.409,6.207,149.296
C05125=1139.574,-22.673,-47.815,179.407,6.206,149.296
C05126=1139.579,-22.923,-47.803,179.404,6.205,149.297
C05127=1139.584,-23.173,-47.790,179.402,6.205,149.297
C05128=1139.590,-23.422,-47.778,179.400,6.204,149.298
C05129=1139.595,-23.672,-47.767,179.397,6.203,149.298
C05130=1139.600,-23.921,-47.755,179.395,6.203,149.299
C05131=1139.605,-24.171,-47.743,179.393,6.202,149.299
C05132=1139.611,-24.441,-47.730,179.390,6.201,149.300
C05133=1139.617,-24.712,-47.716,179.387,6.200,149.301
C05134=1139.622,-24.981,-47.703,179.385,6.199,149.301
C05135=1139.628,-25.251,-47.690,179.382,6.199,149.302
C05136=1139.633,-25.501,-47.678,179.380,6.198,149.302
C05137=1139.639,-25.751,-47.666,179.378,6.197,149.303
C05138=1139.643,-26.000,-47.654,179.375,6.197,149.304
C05139=1139.649,-26.250,-47.643,179.373,6.196,149.304
C05140=1139.654,-26.500,-47.631,179.371,6.195,149.304
C05141=1139.659,-26.749,-47.618,179.368,6.195,149.305
C05142=1139.665,-26.999,-47.606,179.366,6.194,149.306
C05143=1139.669,-27.249,-47.595,179.363,6.194,149.306
C05144=1139.674,-27.498,-47.582,179.361,6.193,149.307
C05145=1139.680,-27.748,-47.570,179.359,6.192,149.307
C05146=1139.685,-27.998,-47.559,179.356,6.192,149.308
C05147=1139.690,-28.247,-47.547,179.353,6.190,149.308
C05148=1139.695,-28.497,-47.535,179.351,6.189,149.309
C05149=1139.701,-28.747,-47.523,179.348,6.189,149.310
C05150=1139.706,-28.997,-47.511,179.346,6.188,149.310
C05151=1139.711,-29.246,-47.500,179.344,6.187,149.311
C05152=1139.716,-29.495,-47.487,179.341,6.187,149.311
C05153=1139.722,-29.745,-47.475,179.339,6.186,149.312
C05154=1139.727,-29.995,-47.464,179.337,6.185,149.312
C05155=1139.732,-30.244,-47.452,179.334,6.185,149.313
C05156=1139.737,-30.494,-47.440,179.332,6.184,149.313
C05157=1139.743,-30.744,-47.428,179.330,6.184,149.314
C05158=1139.747,-30.993,-47.416,179.327,6.183,149.315
C05159=1139.753,-31.243,-47.405,179.325,6.182,149.315
C05160=1139.758,-31.493,-47.393,179.323,6.182,149.316
C05161=1139.763,-31.743,-47.381,179.320,6.181,149.316
C05162=1139.769,-31.992,-47.370,179.318,6.180,149.317
C05163=1139.774,-32.242,-47.358,179.316,6.180,149.317
C05164=1139.779,-32.491,-47.345,179.313,6.179,149.318
C05165=1139.784,-32.741,-47.334,179.311,6.178,149.318
C05166=1139.789,-32.991,-47.322,179.308,6.178,149.319
C05167=1139.794,-33.240,-47.311,179.306,6.177,149.319
C05168=1139.800,-33.490,-47.299,179.304,6.176,149.320
C05169=1139.805,-33.740,-47.287,179.301,6.176,149.321
C05170=1139.810,-33.989,-47.276,179.299,6.175,149.321
C05171=1139.816,-34.239,-47.264,179.297,6.175,149.322
C05172=1139.821,-34.489,-47.252,179.294,6.174,149.322
C05173=1139.826,-34.739,-47.241,179.292,6.173,149.323
C05174=1139.831,-34.989,-47.229,179.290,6.173,149.323
C05175=1139.836,-35.238,-47.218,179.287,6.172,149.324
C05176=1139.842,-35.488,-47.207,179.285,6.171,149.324
C05177=1139.847,-35.738,-47.195,179.283,6.171,149.325
C05178=1139.852,-35.987,-47.183,179.280,6.170,149.326
C05179=1139.858,-36.237,-47.171,179.278,6.169,149.326
C05180=1139.862,-36.487,-47.160,179.275,6.169,149.327
C05181=1139.868,-36.736,-47.149,179.273,6.168,149.327
C05182=1139.874,-36.986,-47.137,179.271,6.167,149.328
C05183=1139.878,-37.235,-47.125,179.268,6.167,149.328
C05184=1139.884,-37.485,-47.114,179.266,6.166,149.329
C05185=1139.889,-37.735,-47.102,179.265,6.166,149.329
C05186=1139.895,-37.984,-47.091,179.262,6.166,149.330
C05187=1139.899,-38.234,-47.079,179.260,6.165,149.331
C05188=1139.905,-38.484,-47.068,179.258,6.164,149.331
C05189=1139.909,-38.733,-47.056,179.255,6.164,149.332
C05190=1139.915,-38.983,-47.044,179.253,6.163,149.332
C05191=1139.920,-39.232,-47.033,179.251,6.162,149.333
C05192=1139.926,-39.482,-47.022,179.248,6.162,149.333
C05193=1139.931,-39.732,-47.010,179.246,6.161,149.334
C05194=1139.936,-39.982,-46.998,179.244,6.160,149.334
C05195=1139.942,-40.232,-46.988,179.241,6.160,149.335
C05196=1139.947,-40.481,-46.976,179.239,6.159,149.336
C05197=1139.952,-40.731,-46.964,179.237,6.158,149.336
C05198=1139.957,-40.981,-46.953,179.234,6.158,149.337
C05199=1139.962,-41.230,-46.942,179.232,6.157,149.337
C05200=1139.968,-41.480,-46.930,179.229,6.156,149.338
C05201=1139.972,-41.729,-46.919,179.227,6.156,149.338
C05202=1139.978,-41.980,-46.908,179.225,6.155,149.339
C05203=1139.983,-42.229,-46.897,179.222,6.154,149.339
C05204=1139.989,-42.479,-46.885,179.220,6.154,149.340
C05205=1139.993,-42.728,-46.874,179.218,6.153,149.340
C05206=1139.999,-42.978,-46.862,179.215,6.152,149.341
C05207=1140.004,-43.228,-46.852,179.213,6.153,149.342
C05208=1140.009,-43.478,-46.840,179.211,6.152,149.342
C05209=1140.015,-43.727,-46.829,179.209,6.151,149.343
C05210=1140.020,-43.976,-46.818,179.206,6.151,149.343
C05211=1140.026,-44.227,-46.806,179.204,6.150,149.344
C05212=1140.030,-44.477,-46.795,179.202,6.149,149.344
C05213=1140.036,-44.725,-46.784,179.199,6.149,149.345
C05214=1140.041,-44.975,-46.772,179.197,6.148,149.345
C05215=1140.046,-45.226,-46.762,179.195,6.147,149.346
C05216=1140.052,-45.475,-46.750,179.192,6.147,149.347
C05217=1140.057,-45.725,-46.739,179.190,6.146,149.347
C05218=1140.062,-45.975,-46.728,179.188,6.145,149.348
C05219=1140.068,-46.224,-46.717,179.185,6.145,149.348
C05220=1140.072,-46.474,-46.706,179.183,6.144,149.349
C05221=1140.077,-46.723,-46.694,179.181,6.144,149.349
C05222=1140.083,-46.973,-46.683,179.179,6.144,149.350
C05223=1140.088,-47.223,-46.672,179.177,6.143,149.350
C05224=1140.093,-47.472,-46.661,179.174,6.142,149.351
C05225=1140.099,-47.722,-46.650,179.172,6.142,149.352
C05226=1140.104,-47.972,-46.639,179.169,6.141,149.352
C05227=1140.109,-48.222,-46.628,179.167,6.140,149.353
C05228=1140.115,-48.471,-46.617,179.165,6.140,149.353
C05229=1140.120,-48.721,-46.605,179.162,6.139,149.354
C05230=1140.125,-48.971,-46.595,179.160,6.138,149.354
C05231=1140.131,-49.220,-46.583,179.158,6.138,149.355
C05232=1140.136,-49.471,-46.573,179.156,6.138,149.355
C05233=1140.141,-49.720,-46.562,179.154,6.137,149.356
C05234=1140.146,-49.969,-46.551,179.151,6.137,149.357
C05235=1140.151,-50.220,-46.539,179.149,6.136,149.357
C05236=1140.158,-50.490,-46.527,179.147,6.135,149.358
C05237=1140.162,-50.761,-46.516,179.144,6.135,149.358
C05238=1140.168,-51.032,-46.504,179.142,6.134,149.359
C05239=1140.174,-51.302,-46.492,179.139,6.134,149.359
C05240=1140.179,-51.552,-46.481,179.137,6.133,149.360
C05241=1140.185,-51.801,-46.470,179.134,6.133,149.361
C05242=1140.190,-52.052,-46.459,179.132,6.132,149.361
C05243=1140.196,-52.301,-46.448,179.130,6.131,149.362
C05244=1140.201,-52.551,-46.438,179.127,6.131,149.362
C05245=1140.205,-52.800,-46.426,179.125,6.130,149.363
C05246=1140.211,-53.050,-46.416,179.123,6.129,149.363
C05247=1140.216,-53.300,-46.404,179.121,6.129,149.364
C05248=1140.222,-53.550,-46.394,179.119,6.129,149.364
C05249=1140.227,-53.799,-46.383,179.116,6.128,149.365
C05250=1140.232,-54.049,-46.372,179.114,6.127,149.365
C05251=1140.237,-54.298,-46.361,179.112,6.127,149.366
C05252=1140.243,-54.549,-46.350,179.109,6.126,149.367
C05253=1140.248,-54.798,-46.339,179.107,6.125,149.367
C05254=1140.253,-55.048,-46.328,179.105,6.125,149.368
C05255=1140.258,-55.298,-46.318,179.103,6.125,149.368
C05256=1140.263,-55.547,-46.307,179.101,6.124,149.369
C05257=1140.269,-55.797,-46.297,179.098,6.124,149.369
C05258=1140.273,-56.046,-46.285,179.096,6.123,149.370
C05259=1140.280,-56.296,-46.275,179.094,6.122,149.370
C05260=1140.285,-56.546,-46.264,179.092,6.121,149.371
C05261=1140.290,-56.795,-46.253,179.089,6.121,149.372
C05262=1140.295,-57.046,-46.243,179.087,6.121,149.372
C05263=1140.301,-57.295,-46.232,179.085,6.120,149.372
C05264=1140.305,-57.545,-46.221,179.082,6.120,149.373
C05265=1140.311,-57.794,-46.211,179.080,6.119,149.374
C05266=1140.316,-58.044,-46.200,179.078,6.118,149.374
C05267=1140.321,-58.294,-46.189,179.075,6.118,149.375
C05268=1140.327,-58.544,-46.178,179.073,6.117,149.375
C05269=1140.332,-58.793,-46.167,179.072,6.117,149.376
C05270=1140.337,-59.043,-46.157,179.069,6.116,149.376
C05271=1140.343,-59.293,-46.147,179.067,6.116,149.377
C05272=1140.348,-59.543,-46.136,179.065,6.115,149.377
C05273=1140.353,-59.792,-46.125,179.062,6.114,149.378
C05274=1140.358,-60.042,-46.114,179.060,6.114,149.379
C05275=1140.364,-60.292,-46.104,179.058,6.113,149.379
C05276=1140.368,-60.541,-46.093,179.056,6.113,149.380
C05277=1140.374,-60.791,-46.083,179.053,6.113,149.380
C05278=1140.379,-61.041,-46.072,179.051,6.112,149.381
C05279=1140.385,-61.291,-46.062,179.049,6.111,149.381
C05280=1140.389,-61.540,-46.051,179.047,6.111,149.382
C05281=1140.395,-61.790,-46.040,179.044,6.110,149.382
C05282=1140.401,-62.039,-46.030,179.042,6.110,149.383
C05283=1140.406,-62.290,-46.020,179.040,6.110,149.383
C05284=1140.411,-62.539,-46.009,179.038,6.109,149.384
C05285=1140.416,-62.789,-45.998,179.035,6.108,149.385
C05286=1140.421,-63.038,-45.988,179.033,6.108,149.385
C05287=1140.426,-63.289,-45.977,179.031,6.107,149.386
C05288=1140.432,-63.538,-45.967,179.029,6.107,149.386
C05289=1140.438,-63.788,-45.957,179.027,6.106,149.387
C05290=1140.443,-64.038,-45.946,179.025,6.106,149.387
C05291=1140.448,-64.287,-45.935,179.022,6.105,149.388
C05292=1140.453,-64.537,-45.925,179.020,6.105,149.388
C05293=1140.459,-64.787,-45.915,179.018,6.105,149.389
C05294=1140.464,-65.036,-45.904,179.016,6.104,149.389
C05295=1140.469,-65.286,-45.894,179.013,6.103,149.390
C05296=1140.475,-65.536,-45.884,179.011,6.103,149.391
C05297=1140.480,-65.786,-45.873,179.009,6.102,149.391
C05298=1140.485,-66.036,-45.863,179.007,6.102,149.392
C05299=1140.491,-66.285,-45.852,179.005,6.102,149.392
C05300=1140.496,-66.535,-45.841,179.002,6.101,149.393
C05301=1140.501,-66.784,-45.831,179.000,6.100,149.393
C05302=1140.505,-67.034,-45.821,178.998,6.100,149.394
C05303=1140.511,-67.284,-45.811,178.995,6.099,149.394
C05304=1140.517,-67.534,-45.801,178.994,6.099,149.395
C05305=1140.522,-67.784,-45.790,178.992,6.098,149.395
C05306=1140.527,-68.033,-45.780,178.989,6.098,149.396
C05307=1140.533,-68.283,-45.770,178.987,6.097,149.397
C05308=1140.538,-68.533,-45.759,178.984,6.096,149.397
C05309=1140.543,-68.783,-45.749,178.983,6.096,149.398
C05310=1140.549,-69.032,-45.739,178.980,6.096,149.398
C05311=1140.553,-69.282,-45.729,178.978,6.095,149.399
C05312=1140.559,-69.532,-45.719,178.976,6.094,149.399
C05313=1140.564,-69.781,-45.708,178.974,6.094,149.400
C05314=1140.569,-70.031,-45.698,178.972,6.094,149.400
C05315=1140.575,-70.281,-45.688,178.969,6.093,149.401
C05316=1140.581,-70.531,-45.677,178.967,6.092,149.401
C05317=1140.586,-70.781,-45.667,178.965,6.092,149.402
C05318=1140.591,-71.030,-45.657,178.963,6.092,149.403
C05319=1140.596,-71.280,-45.647,178.961,6.091,149.403
C05320=1140.601,-71.530,-45.636,178.959,6.091,149.404
C05321=1140.607,-71.779,-45.626,178.956,6.090,149.404
C05322=1140.612,-72.029,-45.616,178.954,6.090,149.405
C05323=1140.618,-72.278,-45.606,178.952,6.089,149.405
C05324=1140.622,-72.528,-45.596,178.950,6.089,149.406
C05325=1140.628,-72.779,-45.586,178.947,6.088,149.406
C05326=1140.634,-73.028,-45.576,178.945,6.088,149.407
C05327=1140.639,-73.278,-45.566,178.943,6.088,149.407
C05328=1140.644,-73.528,-45.555,178.941,6.087,149.408
C05329=1140.649,-73.777,-45.546,178.939,6.086,149.409
C05330=1140.655,-74.027,-45.536,178.936,6.086,149.409
C05331=1140.660,-74.277,-45.525,178.935,6.086,149.409
C05332=1140.665,-74.526,-45.515,178.933,6.085,149.410
C05333=1140.671,-74.776,-45.506,178.930,6.085,149.411
C05334=1140.676,-75.026,-45.496,178.928,6.084,149.411
C05335=1140.681,-75.276,-45.485,178.926,6.084,149.412
C05336=1140.687,-75.526,-45.475,178.924,6.083,149.412
C05337=1140.692,-75.775,-45.465,178.921,6.083,149.413
C05338=1140.697,-76.024,-45.455,178.919,6.082,149.413
C05339=1140.703,-76.275,-45.446,178.918,6.082,149.414
C05340=1140.708,-76.546,-45.435,178.915,6.081,149.414
C05341=1140.714,-76.817,-45.423,178.913,6.081,149.415
C05342=1140.720,-77.089,-45.413,178.910,6.080,149.415
C05343=1140.726,-77.360,-45.402,178.908,6.080,149.416
C05344=1140.730,-77.610,-45.392,178.906,6.079,149.417
C05345=1140.736,-77.860,-45.382,178.903,6.078,149.417
C05346=1140.742,-78.110,-45.372,178.902,6.078,149.418
C05347=1140.747,-78.359,-45.362,178.899,6.078,149.418
C05348=1140.752,-78.609,-45.352,178.897,6.077,149.419
C05349=1140.757,-78.859,-45.342,178.895,6.076,149.419
C05350=1140.763,-79.109,-45.332,178.893,6.076,149.420
C05351=1140.768,-79.358,-45.323,178.890,6.076,149.421
C05352=1140.774,-79.608,-45.312,178.888,6.075,149.421
C05353=1140.780,-79.858,-45.303,178.886,6.074,149.421
C05354=1140.785,-80.107,-45.293,178.884,6.074,149.422
C05355=1140.790,-80.357,-45.283,178.882,6.074,149.422
C05356=1140.795,-80.607,-45.274,178.880,6.073,149.423
C05357=1140.800,-80.857,-45.264,178.878,6.073,149.424
C05358=1140.806,-81.106,-45.253,178.876,6.073,149.424
C05359=1140.811,-81.356,-45.244,178.874,6.072,149.425
C05360=1140.816,-81.607,-45.234,178.871,6.071,149.425
C05361=1140.822,-81.856,-45.224,178.869,6.071,149.426
C05362=1140.827,-82.106,-45.215,178.867,6.071,149.426
C05363=1140.832,-82.355,-45.205,178.865,6.070,149.427
C05364=1140.837,-82.605,-45.195,178.863,6.069,149.427
C05365=1140.843,-82.855,-45.185,178.861,6.070,149.428
C05366=1140.849,-83.104,-45.175,178.859,6.069,149.428
C05367=1140.853,-83.354,-45.165,178.856,6.068,149.429
C05368=1140.859,-83.605,-45.156,178.855,6.068,149.429
C05369=1140.864,-83.854,-45.146,178.852,6.068,149.430
C05370=1140.870,-84.104,-45.137,178.850,6.067,149.431
C05371=1140.875,-84.353,-45.127,178.848,6.066,149.431
C05372=1140.880,-84.603,-45.117,178.846,6.066,149.432
C05373=1140.886,-84.853,-45.107,178.844,6.065,149.432
C05374=1140.891,-85.102,-45.098,178.841,6.065,149.433
C05375=1140.896,-85.353,-45.088,178.840,6.065,149.433
C05376=1140.901,-85.602,-45.078,178.837,6.064,149.434
C05377=1140.907,-85.852,-45.069,178.835,6.064,149.434
C05378=1140.912,-86.102,-45.059,178.834,6.064,149.435
C05379=1140.918,-86.352,-45.050,178.831,6.063,149.435
C05380=1140.923,-86.601,-45.040,178.829,6.063,149.436
C05381=1140.929,-86.851,-45.031,178.827,6.062,149.436
C05382=1140.933,-87.100,-45.021,178.825,6.062,149.437
C05383=1140.939,-87.351,-45.011,178.823,6.061,149.437
C05384=1140.944,-87.600,-45.001,178.820,6.061,149.438
C05385=1140.949,-87.851,-44.992,178.819,6.061,149.439
C05386=1140.954,-88.100,-44.982,178.816,6.060,149.439
C05387=1140.960,-88.350,-44.973,178.814,6.059,149.440
C05388=1140.965,-88.599,-44.963,178.813,6.059,149.440
C05389=1140.971,-88.849,-44.954,178.810,6.059,149.441
C05390=1140.976,-89.099,-44.944,178.808,6.058,149.441
C05391=1140.981,-89.348,-44.935,178.806,6.058,149.442
C05392=1140.987,-89.598,-44.925,178.804,6.057,149.442
C05393=1140.992,-89.848,-44.916,178.802,6.057,149.443
C05394=1140.997,-90.097,-44.906,178.799,6.056,149.443
C05395=1141.003,-90.347,-44.897,178.797,6.056,149.444
C05396=1141.008,-90.597,-44.888,178.795,6.056,149.444
C05397=1141.013,-90.847,-44.878,178.793,6.055,149.445
C05398=1141.019,-91.097,-44.868,178.791,6.055,149.445
C05399=1141.024,-91.346,-44.859,178.789,6.054,149.446
C05400=1141.029,-91.596,-44.850,178.787,6.054,149.446
C05401=1141.035,-91.846,-44.840,178.785,6.054,149.447
C05402=1141.039,-92.096,-44.830,178.783,6.053,149.447
C05403=1141.045,-92.346,-44.821,178.781,6.052,149.448
C05404=1141.050,-92.596,-44.812,178.779,6.052,149.448
C05405=1141.055,-92.845,-44.802,178.777,6.051,149.449
C05406=1141.061,-93.095,-44.793,178.774,6.051,149.450
C05407=1141.066,-93.345,-44.784,178.773,6.051,149.450
C05408=1141.072,-93.595,-44.774,178.770,6.050,149.451
C05409=1141.077,-93.845,-44.765,178.768,6.050,149.451
C05410=1141.082,-94.095,-44.756,178.767,6.050,149.452
C05411=1141.088,-94.344,-44.746,178.764,6.049,149.452
C05412=1141.093,-94.594,-44.737,178.762,6.049,149.453
C05413=1141.098,-94.844,-44.728,178.760,6.049,149.453
C05414=1141.104,-95.093,-44.718,178.758,6.048,149.454
C05415=1141.109,-95.343,-44.709,178.756,6.047,149.454
C05416=1141.115,-95.592,-44.700,178.754,6.047,149.455
C05417=1141.121,-95.842,-44.691,178.752,6.046,149.455
C05418=1141.126,-96.092,-44.681,178.749,6.046,149.456
C05419=1141.131,-96.342,-44.672,178.748,6.046,149.456
C05420=1141.137,-96.592,-44.663,178.745,6.045,149.457
C05421=1141.142,-96.841,-44.653,178.744,6.045,149.457
C05422=1141.147,-97.091,-44.644,178.742,6.045,149.458
C05423=1141.153,-97.341,-44.635,178.739,6.044,149.458
C05424=1141.158,-97.591,-44.626,178.737,6.044,149.459
C05425=1141.163,-97.841,-44.617,178.735,6.043,149.460
C05426=1141.169,-98.090,-44.607,178.733,6.043,149.460
C05427=1141.174,-98.340,-44.598,178.731,6.043,149.460
C05428=1141.179,-98.590,-44.589,178.729,6.042,149.461
C05429=1141.185,-98.840,-44.580,178.727,6.041,149.461
C05430=1141.190,-99.090,-44.571,178.725,6.041,149.462
C05431=1141.195,-99.339,-44.561,178.723,6.041,149.463
C05432=1141.200,-99.589,-44.552,178.720,6.040,149.463
C05433=1141.206,-99.839,-44.543,178.719,6.040,149.464
C05434=1141.212,-100.088,-44.534,178.717,6.039,149.464
C05435=1141.217,-100.338,-44.525,178.715,6.039,149.465
C05436=1141.222,-100.588,-44.516,178.713,6.039,149.465
C05437=1141.228,-100.838,-44.506,178.711,6.038,149.466
C05438=1141.233,-101.087,-44.497,178.709,6.038,149.466
C05439=1141.238,-101.337,-44.488,178.706,6.038,149.467
C05440=1141.243,-101.587,-44.479,178.704,6.037,149.467
C05441=1141.249,-101.837,-44.470,178.703,6.037,149.468
C05442=1141.254,-102.087,-44.461,178.700,6.036,149.468
C05443=1141.259,-102.337,-44.452,178.699,6.036,149.469
C05444=1141.265,-102.608,-44.442,178.696,6.036,149.469
C05445=1141.271,-102.881,-44.433,178.694,6.035,149.470
C05446=1141.277,-103.153,-44.423,178.692,6.034,149.470
C05447=1141.282,-103.425,-44.413,178.690,6.034,149.471
C05448=1141.288,-103.675,-44.404,178.688,6.034,149.472
C05449=1141.294,-103.925,-44.395,178.685,6.033,149.472
C05450=1141.299,-104.175,-44.386,178.684,6.033,149.473
C05451=1141.304,-104.424,-44.377,178.682,6.033,149.473
C05452=1141.310,-104.674,-44.368,178.679,6.032,149.474
C05453=1141.315,-104.924,-44.359,178.678,6.032,149.474
C05454=1141.321,-105.174,-44.350,178.676,6.031,149.475
C05455=1141.326,-105.424,-44.341,178.674,6.031,149.475
C05456=1141.331,-105.674,-44.332,178.671,6.031,149.476
C05457=1141.336,-105.924,-44.323,178.669,6.030,149.476
C05458=1141.342,-106.173,-44.315,178.667,6.030,149.477
C05459=1141.347,-106.423,-44.306,178.665,6.029,149.477
C05460=1141.352,-106.673,-44.297,178.664,6.029,149.478
C05461=1141.358,-106.923,-44.287,178.661,6.029,149.478
C05462=1141.363,-107.173,-44.279,178.659,6.028,149.479
C05463=1141.369,-107.422,-44.270,178.658,6.028,149.479
C05464=1141.374,-107.672,-44.261,178.655,6.027,149.480
C05465=1141.379,-107.921,-44.252,178.653,6.028,149.480
C05466=1141.385,-108.171,-44.243,178.651,6.027,149.481
C05467=1141.390,-108.421,-44.234,178.649,6.026,149.481
C05468=1141.395,-108.671,-44.225,178.647,6.026,149.482
C05469=1141.400,-108.921,-44.217,178.645,6.025,149.482
C05470=1141.406,-109.170,-44.208,178.644,6.025,149.483
C05471=1141.411,-109.420,-44.199,178.641,6.025,149.483
C05472=1141.417,-109.670,-44.190,178.640,6.025,149.484
C05473=1141.422,-109.920,-44.181,178.638,6.024,149.484
C05474=1141.427,-110.170,-44.172,178.635,6.023,149.485
C05475=1141.433,-110.419,-44.164,178.634,6.023,149.485
C05476=1141.439,-110.669,-44.155,178.631,6.023,149.486
